LIN {X -0.064,Y -285.308,Z 785.698,A 0.000,B 0.000,C 90.000,E1 305.598} C_DIS
LIN {X 0.000,Y -296.735,Z 785.683,A 0.000,B 0.000,C 90.000,E1 302.880} C_DIS
LIN {X -0.130,Y -309.503,Z 785.668,A 0.000,B 0.000,C 90.000,E1 300.256} C_DIS
LIN {X -0.044,Y -325.399,Z 785.652,A 0.000,B 0.000,C 90.000,E1 297.334} C_DIS
LIN {X -0.084,Y -344.528,Z 785.634,A 0.000,B 0.000,C 90.000,E1 294.207} C_DIS
LIN {X 0.058,Y -365.735,Z 785.618,A 0.000,B 0.000,C 90.000,E1 291.153} C_DIS
LIN {X 0.141,Y -382.144,Z 785.606,A 0.000,B 0.000,C 90.000,E1 289.087} C_DIS
LIN {X 0.210,Y -399.426,Z 785.595,A 0.000,B 0.000,C 90.000,E1 287.094} C_DIS
LIN {X -0.176,Y -414.390,Z 785.586,A 0.000,B 0.000,C 90.000,E1 285.481} C_DIS
LIN {X 0.184,Y -426.696,Z 785.578,A 0.000,B 0.000,C 90.000,E1 284.064} C_DIS
LIN {X -0.207,Y -438.621,Z 785.571,A 0.000,B 0.000,C 90.000,E1 282.771} C_DIS
LIN {X -0.227,Y -447.840,Z 785.565,A 0.000,B 0.000,C 90.000,E1 281.715} C_DIS
LIN {X -0.140,Y -456.433,Z 785.559,A 0.000,B 0.000,C 90.000,E1 280.658} C_DIS
LIN {X -0.035,Y -464.422,Z 785.553,A 0.000,B 0.000,C 90.000,E1 279.613} C_DIS
LIN {X 0.170,Y -471.836,Z 785.548,A 0.000,B 0.000,C 90.000,E1 278.568} C_DIS
LIN {X 0.131,Y -476.934,Z 785.544,A 0.000,B 0.000,C 90.000,E1 277.814} C_DIS
LIN {X 0.070,Y -481.460,Z 785.539,A 0.000,B 0.000,C 90.000,E1 277.068} C_DIS
LIN {X 0.114,Y -485.271,Z 785.535,A 0.000,B 0.000,C 90.000,E1 276.315} C_DIS
LIN {X 0.133,Y -488.291,Z 785.531,A 0.000,B 0.000,C 90.000,E1 275.568} C_DIS
LIN {X -0.152,Y -489.902,Z 785.528,A 0.000,B 0.000,C 90.000,E1 275.106} C_DIS
LIN {X 0.059,Y -491.124,Z 785.526,A 0.000,B 0.000,C 90.000,E1 274.588} C_DIS
LIN {X -0.247,Y -491.992,Z 785.523,A 0.000,B 0.000,C 90.000,E1 274.131} C_DIS
LIN {X -0.020,Y -492.449,Z 785.520,A 0.000,B 0.000,C 90.000,E1 273.612} C_DIS
LIN {X 0.209,Y -492.461,Z 785.517,A 0.000,B 0.000,C 90.000,E1 273.094} C_DIS
LIN {X -0.078,Y -492.080,Z 785.515,A 0.000,B 0.000,C 90.000,E1 272.636} C_DIS
LIN {X 0.129,Y -491.280,Z 785.512,A 0.000,B 0.000,C 90.000,E1 272.121} C_DIS
LIN {X -0.139,Y -490.046,Z 785.509,A 0.000,B 0.000,C 90.000,E1 271.661} C_DIS
LIN {X 0.060,Y -488.375,Z 785.506,A 0.000,B 0.000,C 90.000,E1 271.146} C_DIS
LIN {X -0.232,Y -486.237,Z 785.504,A 0.000,B 0.000,C 90.000,E1 270.688} C_DIS
LIN {X -0.047,Y -483.535,Z 785.501,A 0.000,B 0.000,C 90.000,E1 270.172} C_DIS
LIN {X 0.118,Y -480.277,Z 785.498,A 0.000,B 0.000,C 90.000,E1 269.656} C_DIS
LIN {X -0.214,Y -476.251,Z 785.495,A 0.000,B 0.000,C 90.000,E1 269.198} C_DIS
LIN {X -0.089,Y -471.307,Z 785.493,A 0.000,B 0.000,C 90.000,E1 268.682} C_DIS
LIN {X 0.184,Y -465.469,Z 785.490,A 0.000,B 0.000,C 90.000,E1 268.167} C_DIS
LIN {X -0.118,Y -462.390,Z 785.489,A 0.000,B 0.000,C 90.000,E1 267.993} C_DIS
LIN {X 0.027,Y -458.873,Z 785.488,A 0.000,B 0.000,C 90.000,E1 267.764} C_DIS
LIN {X 0.008,Y -451.802,Z 785.486,A 0.000,B 0.000,C 90.000,E1 267.421} C_DIS
LIN {X 0.059,Y -444.230,Z 785.484,A 0.000,B 0.000,C 90.000,E1 267.135} C_DIS
LIN {X 0.195,Y -436.200,Z 785.483,A 0.000,B 0.000,C 90.000,E1 266.906} C_DIS
LIN {X 0.089,Y -432.234,Z 785.483,A 0.000,B 0.000,C 90.000,E1 266.846} C_DIS
LIN {X -0.201,Y -423.188,Z 785.482,A 0.000,B 0.000,C 90.000,E1 266.788} C_DIS
LIN {X 0.060,Y -417.117,Z 785.482,A 0.000,B 0.000,C 90.000,E1 266.731} C_DIS
LIN {X -0.009,Y -180.966,Z 785.482,A 0.000,B 0.000,C 90.000,E1 266.731} C_DIS
LIN {X 0.007,Y -180.865,Z 785.472,A 0.000,B 0.000,C 90.000,E1 265.008} C_DIS
LIN {X 0.060,Y -178.978,Z 785.444,A 0.000,B 0.000,C 90.000,E1 259.926} C_DIS
LIN {X 0.069,Y -177.945,Z 785.435,A 0.000,B 0.000,C 90.000,E1 258.229} C_DIS
LIN {X 0.084,Y -175.585,Z 785.411,A 0.000,B 0.000,C 90.000,E1 253.976} C_DIS
LIN {X -0.072,Y -172.311,Z 785.387,A 0.000,B 0.000,C 90.000,E1 249.752} C_DIS
LIN {X -0.093,Y -171.789,Z 785.383,A 0.000,B 0.000,C 90.000,E1 248.901} C_DIS
LIN {X -0.055,Y -169.458,Z 785.368,A 0.000,B 0.000,C 90.000,E1 246.305} C_DIS
LIN {X 0.001,Y -166.786,Z 785.349,A 0.000,B 0.000,C 90.000,E1 242.820} C_DIS
LIN {X -0.003,Y -162.767,Z 785.325,A 0.000,B 0.000,C 90.000,E1 238.456} C_DIS
LIN {X -0.027,Y -161.456,Z 785.315,A 0.000,B 0.000,C 90.000,E1 236.707} C_DIS
LIN {X 0.015,Y -157.450,Z 785.290,A 0.000,B 0.000,C 90.000,E1 232.271} C_DIS
LIN {X -0.053,Y -155.460,Z 785.276,A 0.000,B 0.000,C 90.000,E1 229.622} C_DIS
LIN {X -0.011,Y -151.774,Z 785.251,A 0.000,B 0.000,C 90.000,E1 225.121} C_DIS
LIN {X 0.006,Y -149.980,Z 785.236,A 0.000,B 0.000,C 90.000,E1 222.405} C_DIS
LIN {X -0.074,Y -146.815,Z 785.210,A 0.000,B 0.000,C 90.000,E1 217.890} C_DIS
LIN {X 0.033,Y -145.392,Z 785.195,A 0.000,B 0.000,C 90.000,E1 215.105} C_DIS
LIN {X -0.049,Y -142.828,Z 785.170,A 0.000,B 0.000,C 90.000,E1 210.541} C_DIS
LIN {X 0.007,Y -141.441,Z 785.149,A 0.000,B 0.000,C 90.000,E1 206.821} C_DIS
LIN {X 0.052,Y -139.368,Z 785.113,A 0.000,B 0.000,C 90.000,E1 200.301} C_DIS
LIN {X 0.038,Y -138.815,Z 785.097,A 0.000,B 0.000,C 90.000,E1 197.511} C_DIS
LIN {X -0.048,Y -138.352,Z 785.056,A 0.000,B 0.000,C 90.000,E1 190.074} C_DIS
LIN {X 0.065,Y -139.537,Z 785.004,A 0.000,B 0.000,C 90.000,E1 180.688} C_DIS
LIN {X 0.018,Y -141.227,Z 784.973,A 0.000,B 0.000,C 90.000,E1 175.122} C_DIS
LIN {X -0.023,Y -142.599,Z 784.957,A 0.000,B 0.000,C 90.000,E1 172.356} C_DIS
LIN {X 0.071,Y -144.904,Z 784.932,A 0.000,B 0.000,C 90.000,E1 167.701} C_DIS
LIN {X 0.024,Y -147.533,Z 784.911,A 0.000,B 0.000,C 90.000,E1 164.047} C_DIS
LIN {X -0.044,Y -150.131,Z 784.891,A 0.000,B 0.000,C 90.000,E1 160.423} C_DIS
LIN {X -0.033,Y -153.496,Z 784.871,A 0.000,B 0.000,C 90.000,E1 156.794} C_DIS
LIN {X 0.030,Y -157.861,Z 784.846,A 0.000,B 0.000,C 90.000,E1 152.281} C_DIS
LIN {X -0.014,Y -162.146,Z 784.826,A 0.000,B 0.000,C 90.000,E1 148.742} C_DIS
LIN {X -0.036,Y -166.352,Z 784.807,A 0.000,B 0.000,C 90.000,E1 145.229} C_DIS
LIN {X -0.030,Y -171.368,Z 784.787,A 0.000,B 0.000,C 90.000,E1 141.743} C_DIS
LIN {X -0.103,Y -176.276,Z 784.768,A 0.000,B 0.000,C 90.000,E1 138.324} C_DIS
LIN {X 0.015,Y -180.561,Z 784.754,A 0.000,B 0.000,C 90.000,E1 135.729} C_DIS
LIN {X -0.007,Y -185.963,Z 784.735,A 0.000,B 0.000,C 90.000,E1 132.366} C_DIS
LIN {X 0.050,Y -190.594,Z 784.721,A 0.000,B 0.000,C 90.000,E1 129.850} C_DIS
LIN {X 0.040,Y -192.511,Z 784.715,A 0.000,B 0.000,C 90.000,E1 128.705} C_DIS
LIN {X 0.013,Y -292.777,Z 784.715,A 0.000,B 0.000,C 90.000,E1 128.705} C_DIS
LIN {X -0.041,Y -298.777,Z 784.714,A 0.000,B 0.000,C 90.000,E1 128.463} C_DIS
LIN {X -0.049,Y -301.480,Z 784.712,A 0.000,B 0.000,C 90.000,E1 128.222} C_DIS
LIN {X 0.044,Y -305.237,Z 784.709,A 0.000,B 0.000,C 90.000,E1 127.684} C_DIS
LIN {X -0.001,Y -306.900,Z 784.708,A 0.000,B 0.000,C 90.000,E1 127.363} C_DIS
LIN {X 0.010,Y -308.204,Z 784.706,A 0.000,B 0.000,C 90.000,E1 127.030} C_DIS
LIN {X -0.126,Y -320.271,Z 784.684,A 0.000,B 0.000,C 90.000,E1 123.166} C_DIS
LIN {X 0.162,Y -330.699,Z 784.668,A 0.000,B 0.000,C 90.000,E1 120.256} C_DIS
LIN {X 0.095,Y -342.483,Z 784.653,A 0.000,B 0.000,C 90.000,E1 117.462} C_DIS
LIN {X 0.063,Y -355.724,Z 784.637,A 0.000,B 0.000,C 90.000,E1 114.719} C_DIS
LIN {X 0.022,Y -368.815,Z 784.624,A 0.000,B 0.000,C 90.000,E1 112.333} C_DIS
LIN {X 0.017,Y -383.245,Z 784.611,A 0.000,B 0.000,C 90.000,E1 109.993} C_DIS
LIN {X 0.111,Y -399.118,Z 784.598,A 0.000,B 0.000,C 90.000,E1 107.692} C_DIS
LIN {X -0.026,Y -416.549,Z 784.586,A 0.000,B 0.000,C 90.000,E1 105.481} C_DIS
LIN {X 0.065,Y -435.644,Z 784.574,A 0.000,B 0.000,C 90.000,E1 103.300} C_DIS
LIN {X -0.186,Y -455.766,Z 784.563,A 0.000,B 0.000,C 90.000,E1 101.299} C_DIS
LIN {X 0.127,Y -468.504,Z 784.556,A 0.000,B 0.000,C 90.000,E1 100.074} C_DIS
LIN {X 0.016,Y -470.441,Z 784.555,A 0.000,B 0.000,C 90.000,E1 99.849} C_DIS
LIN {X -0.014,Y -471.912,Z 784.553,A 0.000,B 0.000,C 90.000,E1 99.613} C_DIS
LIN {X 0.087,Y -473.945,Z 784.551,A 0.000,B 0.000,C 90.000,E1 99.095} C_DIS
LIN {X -0.198,Y -474.842,Z 784.548,A 0.000,B 0.000,C 90.000,E1 98.624} C_DIS
LIN {X -0.076,Y -474.760,Z 784.545,A 0.000,B 0.000,C 90.000,E1 98.106} C_DIS
LIN {X 0.054,Y -473.694,Z 784.542,A 0.000,B 0.000,C 90.000,E1 97.587} C_DIS
LIN {X -0.085,Y -472.745,Z 784.541,A 0.000,B 0.000,C 90.000,E1 97.352} C_DIS
LIN {X 0.186,Y -471.459,Z 784.539,A 0.000,B 0.000,C 90.000,E1 97.068} C_DIS
LIN {X -0.107,Y -453.695,Z 784.524,A 0.000,B 0.000,C 90.000,E1 94.302} C_DIS
LIN {X 0.040,Y -443.147,Z 784.514,A 0.000,B 0.000,C 90.000,E1 92.465} C_DIS
LIN {X -0.210,Y -433.992,Z 784.505,A 0.000,B 0.000,C 90.000,E1 90.917} C_DIS
LIN {X -0.191,Y -424.524,Z 784.496,A 0.000,B 0.000,C 90.000,E1 89.312} C_DIS
LIN {X 0.088,Y -414.894,Z 784.487,A 0.000,B 0.000,C 90.000,E1 87.650} C_DIS
LIN {X -0.132,Y -403.562,Z 784.476,A 0.000,B 0.000,C 90.000,E1 85.755} C_DIS
LIN {X -0.143,Y -392.119,Z 784.465,A 0.000,B 0.000,C 90.000,E1 83.799} C_DIS
LIN {X 0.096,Y -376.284,Z 784.450,A 0.000,B 0.000,C 90.000,E1 80.905} C_DIS
LIN {X 0.002,Y -362.489,Z 784.435,A 0.000,B 0.000,C 90.000,E1 78.285} C_DIS
LIN {X 0.095,Y -350.867,Z 784.422,A 0.000,B 0.000,C 90.000,E1 75.880} C_DIS
LIN {X 0.065,Y -339.326,Z 784.408,A 0.000,B 0.000,C 90.000,E1 73.449} C_DIS
LIN {X 0.055,Y -328.066,Z 784.394,A 0.000,B 0.000,C 90.000,E1 70.967} C_DIS
LIN {X -0.107,Y -317.052,Z 784.380,A 0.000,B 0.000,C 90.000,E1 68.465} C_DIS
LIN {X -0.057,Y -302.829,Z 784.360,A 0.000,B 0.000,C 90.000,E1 64.897} C_DIS
LIN {X -0.102,Y -289.904,Z 784.340,A 0.000,B 0.000,C 90.000,E1 61.257} C_DIS
LIN {X -0.056,Y -280.077,Z 784.323,A 0.000,B 0.000,C 90.000,E1 58.201} C_DIS
LIN {X -0.139,Y -271.759,Z 784.308,A 0.000,B 0.000,C 90.000,E1 55.468} C_DIS
LIN {X 0.049,Y -265.658,Z 784.296,A 0.000,B 0.000,C 90.000,E1 53.336} C_DIS
LIN {X -0.092,Y -259.561,Z 784.285,A 0.000,B 0.000,C 90.000,E1 51.251} C_DIS
LIN {X 0.013,Y -251.506,Z 784.269,A 0.000,B 0.000,C 90.000,E1 48.366} C_DIS
LIN {X -0.117,Y -241.907,Z 784.248,A 0.000,B 0.000,C 90.000,E1 44.757} C_DIS
LIN {X -0.069,Y -236.363,Z 784.236,A 0.000,B 0.000,C 90.000,E1 42.528} C_DIS
LIN {X 0.039,Y -227.342,Z 784.215,A 0.000,B 0.000,C 90.000,E1 38.749} C_DIS
LIN {X -0.030,Y -218.837,Z 784.194,A 0.000,B 0.000,C 90.000,E1 34.945} C_DIS
LIN {X -0.017,Y -211.028,Z 784.172,A 0.000,B 0.000,C 90.000,E1 31.052} C_DIS
LIN {X -0.029,Y -205.490,Z 784.155,A 0.000,B 0.000,C 90.000,E1 27.897} C_DIS
LIN {X -0.006,Y -200.725,Z 784.137,A 0.000,B 0.000,C 90.000,E1 24.695} C_DIS
LIN {X -0.035,Y -195.745,Z 784.115,A 0.000,B 0.000,C 90.000,E1 20.663} C_DIS
LIN {X 0.009,Y -191.908,Z 784.092,A 0.000,B 0.000,C 90.000,E1 16.567} C_DIS
LIN {X -0.103,Y -188.694,Z 784.065,A 0.000,B 0.000,C 90.000,E1 11.658} C_DIS
LIN {X 0.003,Y -186.624,Z 784.018,A 0.000,B 0.000,C 90.000,E1 3.326} C_DIS
LIN {X 0.001,Y -188.497,Z 783.970,A 0.000,B 0.000,C 90.000,E1 354.546} C_DIS
LIN {X 0.004,Y -192.032,Z 783.938,A 0.000,B 0.000,C 90.000,E1 348.757} C_DIS
LIN {X 0.089,Y -195.633,Z 783.915,A 0.000,B 0.000,C 90.000,E1 344.629} C_DIS
LIN {X -0.062,Y -200.258,Z 783.892,A 0.000,B 0.000,C 90.000,E1 340.604} C_DIS
LIN {X 0.083,Y -205.972,Z 783.870,A 0.000,B 0.000,C 90.000,E1 336.538} C_DIS
LIN {X -0.024,Y -211.217,Z 783.852,A 0.000,B 0.000,C 90.000,E1 333.384} C_DIS
LIN {X -0.038,Y -218.499,Z 783.830,A 0.000,B 0.000,C 90.000,E1 329.459} C_DIS
LIN {X 0.036,Y -224.827,Z 783.813,A 0.000,B 0.000,C 90.000,E1 326.342} C_DIS
LIN {X -0.086,Y -233.389,Z 783.792,A 0.000,B 0.000,C 90.000,E1 322.557} C_DIS
LIN {X 0.078,Y -242.712,Z 783.771,A 0.000,B 0.000,C 90.000,E1 318.771} C_DIS
LIN {X -0.015,Y -252.902,Z 783.751,A 0.000,B 0.000,C 90.000,E1 315.121} C_DIS
LIN {X 0.002,Y -262.764,Z 783.733,A 0.000,B 0.000,C 90.000,E1 311.881} C_DIS
LIN {X -0.116,Y -274.750,Z 783.713,A 0.000,B 0.000,C 90.000,E1 308.382} C_DIS
LIN {X 0.093,Y -288.032,Z 783.694,A 0.000,B 0.000,C 90.000,E1 304.898} C_DIS
LIN {X 0.064,Y -298.190,Z 783.681,A 0.000,B 0.000,C 90.000,E1 302.546} C_DIS
LIN {X -0.026,Y -311.133,Z 783.666,A 0.000,B 0.000,C 90.000,E1 299.922} C_DIS
LIN {X 0.119,Y -327.130,Z 783.650,A 0.000,B 0.000,C 90.000,E1 297.001} C_DIS
LIN {X -0.012,Y -344.443,Z 783.634,A 0.000,B 0.000,C 90.000,E1 294.207} C_DIS
LIN {X 0.070,Y -363.354,Z 783.619,A 0.000,B 0.000,C 90.000,E1 291.461} C_DIS
LIN {X 0.060,Y -379.537,Z 783.608,A 0.000,B 0.000,C 90.000,E1 289.396} C_DIS
LIN {X 0.094,Y -399.416,Z 783.595,A 0.000,B 0.000,C 90.000,E1 287.094} C_DIS
LIN {X 0.035,Y -414.432,Z 783.586,A 0.000,B 0.000,C 90.000,E1 285.426} C_DIS
LIN {X 0.047,Y -426.654,Z 783.578,A 0.000,B 0.000,C 90.000,E1 284.064} C_DIS
LIN {X 0.079,Y -438.510,Z 783.571,A 0.000,B 0.000,C 90.000,E1 282.715} C_DIS
LIN {X 0.066,Y -447.727,Z 783.565,A 0.000,B 0.000,C 90.000,E1 281.658} C_DIS
LIN {X 0.159,Y -456.331,Z 783.559,A 0.000,B 0.000,C 90.000,E1 280.602} C_DIS
LIN {X -0.189,Y -464.285,Z 783.553,A 0.000,B 0.000,C 90.000,E1 279.613} C_DIS
LIN {X 0.012,Y -471.747,Z 783.548,A 0.000,B 0.000,C 90.000,E1 278.568} C_DIS
LIN {X -0.237,Y -478.485,Z 783.542,A 0.000,B 0.000,C 90.000,E1 277.587} C_DIS
LIN {X -0.221,Y -482.779,Z 783.538,A 0.000,B 0.000,C 90.000,E1 276.834} C_DIS
LIN {X -0.229,Y -486.319,Z 783.534,A 0.000,B 0.000,C 90.000,E1 276.087} C_DIS
LIN {X -0.033,Y -488.289,Z 783.531,A 0.000,B 0.000,C 90.000,E1 275.568} C_DIS
LIN {X 0.169,Y -489.900,Z 783.528,A 0.000,B 0.000,C 90.000,E1 275.049} C_DIS
LIN {X -0.107,Y -491.132,Z 783.525,A 0.000,B 0.000,C 90.000,E1 274.588} C_DIS
LIN {X 0.077,Y -491.995,Z 783.523,A 0.000,B 0.000,C 90.000,E1 274.073} C_DIS
LIN {X -0.187,Y -492.450,Z 783.520,A 0.000,B 0.000,C 90.000,E1 273.612} C_DIS
LIN {X 0.042,Y -492.493,Z 783.517,A 0.000,B 0.000,C 90.000,E1 273.094} C_DIS
LIN {X 0.246,Y -492.142,Z 783.514,A 0.000,B 0.000,C 90.000,E1 272.579} C_DIS
LIN {X -0.038,Y -491.332,Z 783.512,A 0.000,B 0.000,C 90.000,E1 272.121} C_DIS
LIN {X 0.184,Y -490.093,Z 783.509,A 0.000,B 0.000,C 90.000,E1 271.604} C_DIS
LIN {X -0.104,Y -488.417,Z 783.506,A 0.000,B 0.000,C 90.000,E1 271.146} C_DIS
LIN {X 0.090,Y -486.263,Z 783.504,A 0.000,B 0.000,C 90.000,E1 270.630} C_DIS
LIN {X -0.210,Y -483.566,Z 783.501,A 0.000,B 0.000,C 90.000,E1 270.172} C_DIS
LIN {X -0.044,Y -480.305,Z 783.498,A 0.000,B 0.000,C 90.000,E1 269.656} C_DIS
LIN {X 0.102,Y -476.248,Z 783.495,A 0.000,B 0.000,C 90.000,E1 269.141} C_DIS
LIN {X -0.073,Y -473.928,Z 783.494,A 0.000,B 0.000,C 90.000,E1 268.912} C_DIS
LIN {X 0.158,Y -468.582,Z 783.491,A 0.000,B 0.000,C 90.000,E1 268.396} C_DIS
LIN {X 0.107,Y -465.525,Z 783.490,A 0.000,B 0.000,C 90.000,E1 268.165} C_DIS
LIN {X -0.198,Y -462.443,Z 783.489,A 0.000,B 0.000,C 90.000,E1 267.993} C_DIS
LIN {X -0.033,Y -455.738,Z 783.487,A 0.000,B 0.000,C 90.000,E1 267.593} C_DIS
LIN {X -0.218,Y -448.581,Z 783.485,A 0.000,B 0.000,C 90.000,E1 267.306} C_DIS
LIN {X 0.097,Y -440.943,Z 783.484,A 0.000,B 0.000,C 90.000,E1 267.020} C_DIS
LIN {X 0.036,Y -432.403,Z 783.482,A 0.000,B 0.000,C 90.000,E1 266.846} C_DIS
LIN {X 0.149,Y -423.558,Z 783.482,A 0.000,B 0.000,C 90.000,E1 266.731} C_DIS
LIN {X -0.020,Y -418.188,Z 783.482,A 0.000,B 0.000,C 90.000,E1 266.731} C_DIS
LIN {X -0.045,Y -180.965,Z 783.482,A 0.000,B 0.000,C 90.000,E1 266.731} C_DIS
LIN {X -0.035,Y -180.861,Z 783.472,A 0.000,B 0.000,C 90.000,E1 265.008} C_DIS
LIN {X 0.019,Y -178.974,Z 783.444,A 0.000,B 0.000,C 90.000,E1 259.926} C_DIS
LIN {X 0.029,Y -177.936,Z 783.435,A 0.000,B 0.000,C 90.000,E1 258.229} C_DIS
LIN {X 0.044,Y -175.575,Z 783.411,A 0.000,B 0.000,C 90.000,E1 253.976} C_DIS
LIN {X 0.051,Y -172.303,Z 783.387,A 0.000,B 0.000,C 90.000,E1 249.699} C_DIS
LIN {X 0.028,Y -171.781,Z 783.383,A 0.000,B 0.000,C 90.000,E1 248.847} C_DIS
LIN {X 0.000,Y -168.712,Z 783.363,A 0.000,B 0.000,C 90.000,E1 245.409} C_DIS
LIN {X 0.039,Y -166.776,Z 783.349,A 0.000,B 0.000,C 90.000,E1 242.794} C_DIS
LIN {X -0.041,Y -162.756,Z 783.325,A 0.000,B 0.000,C 90.000,E1 238.456} C_DIS
LIN {X -0.065,Y -161.446,Z 783.315,A 0.000,B 0.000,C 90.000,E1 236.707} C_DIS
LIN {X -0.024,Y -157.439,Z 783.290,A 0.000,B 0.000,C 90.000,E1 232.271} C_DIS
LIN {X 0.011,Y -155.447,Z 783.276,A 0.000,B 0.000,C 90.000,E1 229.585} C_DIS
LIN {X 0.059,Y -151.766,Z 783.251,A 0.000,B 0.000,C 90.000,E1 225.081} C_DIS
LIN {X 0.070,Y -149.968,Z 783.236,A 0.000,B 0.000,C 90.000,E1 222.366} C_DIS
LIN {X -0.019,Y -146.806,Z 783.210,A 0.000,B 0.000,C 90.000,E1 217.855} C_DIS
LIN {X -0.003,Y -145.383,Z 783.195,A 0.000,B 0.000,C 90.000,E1 215.105} C_DIS
LIN {X -0.011,Y -142.442,Z 783.164,A 0.000,B 0.000,C 90.000,E1 209.589} C_DIS
LIN {X 0.036,Y -141.434,Z 783.149,A 0.000,B 0.000,C 90.000,E1 206.796} C_DIS
LIN {X 0.017,Y -139.366,Z 783.113,A 0.000,B 0.000,C 90.000,E1 200.301} C_DIS
LIN {X 0.003,Y -138.813,Z 783.097,A 0.000,B 0.000,C 90.000,E1 197.511} C_DIS
LIN {X 0.054,Y -138.351,Z 783.056,A 0.000,B 0.000,C 90.000,E1 190.018} C_DIS
LIN {X 0.030,Y -139.539,Z 783.004,A 0.000,B 0.000,C 90.000,E1 180.688} C_DIS
LIN {X -0.018,Y -141.233,Z 782.973,A 0.000,B 0.000,C 90.000,E1 175.122} C_DIS
LIN {X -0.059,Y -142.604,Z 782.957,A 0.000,B 0.000,C 90.000,E1 172.356} C_DIS
LIN {X 0.035,Y -144.913,Z 782.932,A 0.000,B 0.000,C 90.000,E1 167.701} C_DIS
LIN {X 0.028,Y -147.542,Z 782.911,A 0.000,B 0.000,C 90.000,E1 164.031} C_DIS
LIN {X 0.061,Y -150.143,Z 782.891,A 0.000,B 0.000,C 90.000,E1 160.369} C_DIS
LIN {X -0.070,Y -153.511,Z 782.871,A 0.000,B 0.000,C 90.000,E1 156.794} C_DIS
LIN {X -0.007,Y -157.876,Z 782.846,A 0.000,B 0.000,C 90.000,E1 152.281} C_DIS
LIN {X -0.052,Y -162.163,Z 782.826,A 0.000,B 0.000,C 90.000,E1 148.742} C_DIS
LIN {X 0.062,Y -166.369,Z 782.807,A 0.000,B 0.000,C 90.000,E1 145.182} C_DIS
LIN {X 0.065,Y -171.386,Z 782.787,A 0.000,B 0.000,C 90.000,E1 141.698} C_DIS
LIN {X 0.105,Y -176.296,Z 782.768,A 0.000,B 0.000,C 90.000,E1 138.243} C_DIS
LIN {X -0.027,Y -180.583,Z 782.754,A 0.000,B 0.000,C 90.000,E1 135.729} C_DIS
LIN {X -0.048,Y -185.985,Z 782.735,A 0.000,B 0.000,C 90.000,E1 132.366} C_DIS
LIN {X 0.007,Y -190.619,Z 782.721,A 0.000,B 0.000,C 90.000,E1 129.850} C_DIS
LIN {X -0.066,Y -192.489,Z 782.715,A 0.000,B 0.000,C 90.000,E1 128.749} C_DIS
LIN {X -0.136,Y -292.326,Z 782.715,A 0.000,B 0.000,C 90.000,E1 128.749} C_DIS
LIN {X 0.085,Y -294.367,Z 782.715,A 0.000,B 0.000,C 90.000,E1 128.669} C_DIS
LIN {X -0.106,Y -299.048,Z 782.714,A 0.000,B 0.000,C 90.000,E1 128.463} C_DIS
LIN {X 0.122,Y -301.653,Z 782.712,A 0.000,B 0.000,C 90.000,E1 128.177} C_DIS
LIN {X 0.079,Y -305.413,Z 782.709,A 0.000,B 0.000,C 90.000,E1 127.649} C_DIS
LIN {X 0.090,Y -307.024,Z 782.707,A 0.000,B 0.000,C 90.000,E1 127.317} C_DIS
LIN {X 0.043,Y -308.289,Z 782.706,A 0.000,B 0.000,C 90.000,E1 126.996} C_DIS
LIN {X 0.162,Y -320.344,Z 782.684,A 0.000,B 0.000,C 90.000,E1 123.086} C_DIS
LIN {X 0.005,Y -330.785,Z 782.668,A 0.000,B 0.000,C 90.000,E1 120.256} C_DIS
LIN {X -0.066,Y -342.583,Z 782.653,A 0.000,B 0.000,C 90.000,E1 117.462} C_DIS
LIN {X -0.102,Y -355.838,Z 782.637,A 0.000,B 0.000,C 90.000,E1 114.719} C_DIS
LIN {X -0.146,Y -368.942,Z 782.624,A 0.000,B 0.000,C 90.000,E1 112.333} C_DIS
LIN {X -0.154,Y -383.387,Z 782.611,A 0.000,B 0.000,C 90.000,E1 109.993} C_DIS
LIN {X -0.063,Y -399.278,Z 782.598,A 0.000,B 0.000,C 90.000,E1 107.692} C_DIS
LIN {X 0.197,Y -416.726,Z 782.586,A 0.000,B 0.000,C 90.000,E1 105.426} C_DIS
LIN {X -0.115,Y -435.837,Z 782.574,A 0.000,B 0.000,C 90.000,E1 103.300} C_DIS
LIN {X 0.086,Y -455.967,Z 782.563,A 0.000,B 0.000,C 90.000,E1 101.243} C_DIS
LIN {X -0.044,Y -468.675,Z 782.556,A 0.000,B 0.000,C 90.000,E1 100.074} C_DIS
LIN {X -0.170,Y -470.586,Z 782.555,A 0.000,B 0.000,C 90.000,E1 99.849} C_DIS
LIN {X -0.217,Y -472.037,Z 782.553,A 0.000,B 0.000,C 90.000,E1 99.613} C_DIS
LIN {X -0.116,Y -474.018,Z 782.550,A 0.000,B 0.000,C 90.000,E1 99.095} C_DIS
LIN {X 0.069,Y -474.873,Z 782.548,A 0.000,B 0.000,C 90.000,E1 98.568} C_DIS
LIN {X 0.192,Y -474.754,Z 782.545,A 0.000,B 0.000,C 90.000,E1 98.049} C_DIS
LIN {X -0.146,Y -473.645,Z 782.542,A 0.000,B 0.000,C 90.000,E1 97.587} C_DIS
LIN {X 0.184,Y -472.671,Z 782.541,A 0.000,B 0.000,C 90.000,E1 97.296} C_DIS
LIN {X -0.015,Y -471.355,Z 782.539,A 0.000,B 0.000,C 90.000,E1 97.068} C_DIS
LIN {X 0.150,Y -453.580,Z 782.524,A 0.000,B 0.000,C 90.000,E1 94.245} C_DIS
LIN {X -0.153,Y -443.023,Z 782.514,A 0.000,B 0.000,C 90.000,E1 92.465} C_DIS
LIN {X 0.032,Y -433.887,Z 782.505,A 0.000,B 0.000,C 90.000,E1 90.859} C_DIS
LIN {X 0.044,Y -424.425,Z 782.496,A 0.000,B 0.000,C 90.000,E1 89.255} C_DIS
LIN {X -0.006,Y -413.178,Z 782.485,A 0.000,B 0.000,C 90.000,E1 87.364} C_DIS
LIN {X 0.087,Y -403.472,Z 782.476,A 0.000,B 0.000,C 90.000,E1 85.698} C_DIS
LIN {X 0.077,Y -390.407,Z 782.464,A 0.000,B 0.000,C 90.000,E1 83.457} C_DIS
LIN {X -0.079,Y -376.210,Z 782.449,A 0.000,B 0.000,C 90.000,E1 80.905} C_DIS
LIN {X 0.162,Y -360.948,Z 782.433,A 0.000,B 0.000,C 90.000,E1 77.937} C_DIS
LIN {X -0.045,Y -349.388,Z 782.420,A 0.000,B 0.000,C 90.000,E1 75.574} C_DIS
LIN {X -0.098,Y -337.880,Z 782.406,A 0.000,B 0.000,C 90.000,E1 73.142} C_DIS
LIN {X 0.178,Y -326.659,Z 782.392,A 0.000,B 0.000,C 90.000,E1 70.604} C_DIS
LIN {X -0.095,Y -314.404,Z 782.377,A 0.000,B 0.000,C 90.000,E1 67.794} C_DIS
LIN {X -0.012,Y -300.461,Z 782.357,A 0.000,B 0.000,C 90.000,E1 64.204} C_DIS
LIN {X -0.009,Y -287.816,Z 782.336,A 0.000,B 0.000,C 90.000,E1 60.539} C_DIS
LIN {X 0.135,Y -278.207,Z 782.319,A 0.000,B 0.000,C 90.000,E1 57.454} C_DIS
LIN {X 0.152,Y -269.987,Z 782.304,A 0.000,B 0.000,C 90.000,E1 54.689} C_DIS
LIN {X 0.059,Y -261.882,Z 782.288,A 0.000,B 0.000,C 90.000,E1 51.904} C_DIS
LIN {X 0.053,Y -253.846,Z 782.273,A 0.000,B 0.000,C 90.000,E1 49.057} C_DIS
LIN {X -0.001,Y -244.130,Z 782.253,A 0.000,B 0.000,C 90.000,E1 45.445} C_DIS
LIN {X -0.133,Y -236.699,Z 782.236,A 0.000,B 0.000,C 90.000,E1 42.528} C_DIS
LIN {X -0.012,Y -227.656,Z 782.215,A 0.000,B 0.000,C 90.000,E1 38.749} C_DIS
LIN {X -0.071,Y -219.130,Z 782.194,A 0.000,B 0.000,C 90.000,E1 34.945} C_DIS
LIN {X -0.048,Y -211.314,Z 782.172,A 0.000,B 0.000,C 90.000,E1 31.052} C_DIS
LIN {X -0.051,Y -205.757,Z 782.155,A 0.000,B 0.000,C 90.000,E1 27.897} C_DIS
LIN {X -0.045,Y -199.916,Z 782.133,A 0.000,B 0.000,C 90.000,E1 23.898} C_DIS
LIN {X 0.090,Y -195.141,Z 782.110,A 0.000,B 0.000,C 90.000,E1 19.812} C_DIS
LIN {X 0.058,Y -191.502,Z 782.088,A 0.000,B 0.000,C 90.000,E1 15.733} C_DIS
LIN {X 0.072,Y -188.523,Z 782.060,A 0.000,B 0.000,C 90.000,E1 10.782} C_DIS
LIN {X -0.029,Y -187.969,Z 781.979,A 0.000,B 0.000,C 90.000,E1 356.216} C_DIS
LIN {X 0.080,Y -190.984,Z 781.947,A 0.000,B 0.000,C 90.000,E1 350.387} C_DIS
LIN {X 0.049,Y -194.962,Z 781.919,A 0.000,B 0.000,C 90.000,E1 345.463} C_DIS
LIN {X 0.002,Y -199.392,Z 781.897,A 0.000,B 0.000,C 90.000,E1 341.402} C_DIS
LIN {X 0.040,Y -204.919,Z 781.874,A 0.000,B 0.000,C 90.000,E1 337.358} C_DIS
LIN {X 0.095,Y -209.981,Z 781.857,A 0.000,B 0.000,C 90.000,E1 334.152} C_DIS
LIN {X -0.060,Y -217.120,Z 781.835,A 0.000,B 0.000,C 90.000,E1 330.255} C_DIS
LIN {X 0.045,Y -223.348,Z 781.817,A 0.000,B 0.000,C 90.000,E1 327.120} C_DIS
LIN {X 0.057,Y -231.725,Z 781.796,A 0.000,B 0.000,C 90.000,E1 323.290} C_DIS
LIN {X 0.013,Y -240.884,Z 781.775,A 0.000,B 0.000,C 90.000,E1 319.542} C_DIS
LIN {X 0.036,Y -249.821,Z 781.757,A 0.000,B 0.000,C 90.000,E1 316.215} C_DIS
LIN {X -0.004,Y -260.516,Z 781.737,A 0.000,B 0.000,C 90.000,E1 312.609} C_DIS
LIN {X -0.012,Y -272.284,Z 781.717,A 0.000,B 0.000,C 90.000,E1 309.072} C_DIS
LIN {X -0.005,Y -282.531,Z 781.702,A 0.000,B 0.000,C 90.000,E1 306.297} C_DIS
LIN {X 0.134,Y -296.607,Z 781.683,A 0.000,B 0.000,C 90.000,E1 302.880} C_DIS
LIN {X 0.006,Y -309.381,Z 781.668,A 0.000,B 0.000,C 90.000,E1 300.256} C_DIS
LIN {X -0.104,Y -327.052,Z 781.650,A 0.000,B 0.000,C 90.000,E1 297.052} C_DIS
LIN {X 0.065,Y -342.333,Z 781.636,A 0.000,B 0.000,C 90.000,E1 294.515} C_DIS
LIN {X 0.141,Y -363.209,Z 781.619,A 0.000,B 0.000,C 90.000,E1 291.461} C_DIS
LIN {X 0.002,Y -384.028,Z 781.605,A 0.000,B 0.000,C 90.000,E1 288.852} C_DIS
LIN {X -0.084,Y -398.989,Z 781.595,A 0.000,B 0.000,C 90.000,E1 287.149} C_DIS
LIN {X -0.159,Y -414.006,Z 781.586,A 0.000,B 0.000,C 90.000,E1 285.481} C_DIS
LIN {X 0.213,Y -426.245,Z 781.578,A 0.000,B 0.000,C 90.000,E1 284.064} C_DIS
LIN {X -0.184,Y -438.092,Z 781.571,A 0.000,B 0.000,C 90.000,E1 282.771} C_DIS
LIN {X -0.208,Y -447.272,Z 781.565,A 0.000,B 0.000,C 90.000,E1 281.715} C_DIS
LIN {X -0.128,Y -455.916,Z 781.559,A 0.000,B 0.000,C 90.000,E1 280.658} C_DIS
LIN {X -0.197,Y -465.788,Z 781.552,A 0.000,B 0.000,C 90.000,E1 279.378} C_DIS
LIN {X -0.051,Y -473.158,Z 781.546,A 0.000,B 0.000,C 90.000,E1 278.341} C_DIS
LIN {X -0.082,Y -478.155,Z 781.542,A 0.000,B 0.000,C 90.000,E1 277.587} C_DIS
LIN {X -0.068,Y -482.519,Z 781.538,A 0.000,B 0.000,C 90.000,E1 276.834} C_DIS
LIN {X -0.076,Y -486.141,Z 781.534,A 0.000,B 0.000,C 90.000,E1 276.087} C_DIS
LIN {X 0.119,Y -488.156,Z 781.531,A 0.000,B 0.000,C 90.000,E1 275.568} C_DIS
LIN {X -0.167,Y -489.796,Z 781.528,A 0.000,B 0.000,C 90.000,E1 275.106} C_DIS
LIN {X 0.044,Y -491.057,Z 781.526,A 0.000,B 0.000,C 90.000,E1 274.588} C_DIS
LIN {X 0.227,Y -491.967,Z 781.523,A 0.000,B 0.000,C 90.000,E1 274.073} C_DIS
LIN {X -0.037,Y -492.450,Z 781.520,A 0.000,B 0.000,C 90.000,E1 273.612} C_DIS
LIN {X 0.192,Y -492.545,Z 781.517,A 0.000,B 0.000,C 90.000,E1 273.094} C_DIS
LIN {X -0.096,Y -492.202,Z 781.515,A 0.000,B 0.000,C 90.000,E1 272.636} C_DIS
LIN {X 0.113,Y -491.452,Z 781.512,A 0.000,B 0.000,C 90.000,E1 272.121} C_DIS
LIN {X -0.156,Y -490.242,Z 781.509,A 0.000,B 0.000,C 90.000,E1 271.661} C_DIS
LIN {X 0.046,Y -488.584,Z 781.506,A 0.000,B 0.000,C 90.000,E1 271.146} C_DIS
LIN {X 0.241,Y -486.490,Z 781.504,A 0.000,B 0.000,C 90.000,E1 270.630} C_DIS
LIN {X -0.059,Y -483.827,Z 781.501,A 0.000,B 0.000,C 90.000,E1 270.172} C_DIS
LIN {X 0.106,Y -480.578,Z 781.498,A 0.000,B 0.000,C 90.000,E1 269.656} C_DIS
LIN {X -0.223,Y -476.518,Z 781.495,A 0.000,B 0.000,C 90.000,E1 269.198} C_DIS
LIN {X 0.078,Y -474.281,Z 781.494,A 0.000,B 0.000,C 90.000,E1 268.912} C_DIS
LIN {X -0.164,Y -468.975,Z 781.491,A 0.000,B 0.000,C 90.000,E1 268.453} C_DIS
LIN {X -0.232,Y -465.939,Z 781.490,A 0.000,B 0.000,C 90.000,E1 268.224} C_DIS
LIN {X 0.079,Y -459.451,Z 781.488,A 0.000,B 0.000,C 90.000,E1 267.764} C_DIS
LIN {X 0.044,Y -456.199,Z 781.487,A 0.000,B 0.000,C 90.000,E1 267.593} C_DIS
LIN {X -0.194,Y -449.007,Z 781.485,A 0.000,B 0.000,C 90.000,E1 267.306} C_DIS
LIN {X 0.096,Y -441.420,Z 781.484,A 0.000,B 0.000,C 90.000,E1 267.020} C_DIS
LIN {X 0.139,Y -437.039,Z 781.483,A 0.000,B 0.000,C 90.000,E1 266.906} C_DIS
LIN {X -0.149,Y -427.197,Z 781.482,A 0.000,B 0.000,C 90.000,E1 266.788} C_DIS
LIN {X -0.115,Y -418.313,Z 781.482,A 0.000,B 0.000,C 90.000,E1 266.731} C_DIS
LIN {X -0.068,Y -180.964,Z 781.482,A 0.000,B 0.000,C 90.000,E1 266.731} C_DIS
LIN {X -0.062,Y -180.859,Z 781.472,A 0.000,B 0.000,C 90.000,E1 265.008} C_DIS
LIN {X -0.008,Y -178.972,Z 781.444,A 0.000,B 0.000,C 90.000,E1 259.926} C_DIS
LIN {X 0.002,Y -177.930,Z 781.435,A 0.000,B 0.000,C 90.000,E1 258.229} C_DIS
LIN {X 0.017,Y -175.569,Z 781.411,A 0.000,B 0.000,C 90.000,E1 253.976} C_DIS
LIN {X 0.024,Y -172.297,Z 781.387,A 0.000,B 0.000,C 90.000,E1 249.699} C_DIS
LIN {X 0.001,Y -171.775,Z 781.383,A 0.000,B 0.000,C 90.000,E1 248.847} C_DIS
LIN {X -0.026,Y -168.704,Z 781.363,A 0.000,B 0.000,C 90.000,E1 245.409} C_DIS
LIN {X 0.013,Y -166.769,Z 781.349,A 0.000,B 0.000,C 90.000,E1 242.794} C_DIS
LIN {X 0.071,Y -162.749,Z 781.325,A 0.000,B 0.000,C 90.000,E1 238.408} C_DIS
LIN {X -0.091,Y -161.439,Z 781.315,A 0.000,B 0.000,C 90.000,E1 236.707} C_DIS
LIN {X -0.049,Y -157.432,Z 781.290,A 0.000,B 0.000,C 90.000,E1 232.271} C_DIS
LIN {X -0.014,Y -155.438,Z 781.275,A 0.000,B 0.000,C 90.000,E1 229.585} C_DIS
LIN {X 0.034,Y -151.759,Z 781.251,A 0.000,B 0.000,C 90.000,E1 225.081} C_DIS
LIN {X 0.046,Y -149.960,Z 781.235,A 0.000,B 0.000,C 90.000,E1 222.366} C_DIS
LIN {X 0.073,Y -146.802,Z 781.210,A 0.000,B 0.000,C 90.000,E1 217.810} C_DIS
LIN {X -0.027,Y -145.377,Z 781.195,A 0.000,B 0.000,C 90.000,E1 215.105} C_DIS
LIN {X -0.034,Y -142.439,Z 781.164,A 0.000,B 0.000,C 90.000,E1 209.589} C_DIS
LIN {X 0.013,Y -141.429,Z 781.149,A 0.000,B 0.000,C 90.000,E1 206.796} C_DIS
LIN {X -0.006,Y -139.365,Z 781.113,A 0.000,B 0.000,C 90.000,E1 200.301} C_DIS
LIN {X -0.020,Y -138.810,Z 781.097,A 0.000,B 0.000,C 90.000,E1 197.511} C_DIS
LIN {X 0.030,Y -138.351,Z 781.056,A 0.000,B 0.000,C 90.000,E1 190.018} C_DIS
LIN {X 0.007,Y -139.541,Z 781.004,A 0.000,B 0.000,C 90.000,E1 180.688} C_DIS
LIN {X -0.041,Y -141.237,Z 780.973,A 0.000,B 0.000,C 90.000,E1 175.122} C_DIS
LIN {X 0.059,Y -142.608,Z 780.957,A 0.000,B 0.000,C 90.000,E1 172.299} C_DIS
LIN {X 0.012,Y -144.919,Z 780.932,A 0.000,B 0.000,C 90.000,E1 167.701} C_DIS
LIN {X 0.004,Y -147.548,Z 780.911,A 0.000,B 0.000,C 90.000,E1 164.031} C_DIS
LIN {X 0.036,Y -150.151,Z 780.891,A 0.000,B 0.000,C 90.000,E1 160.369} C_DIS
LIN {X 0.046,Y -153.520,Z 780.871,A 0.000,B 0.000,C 90.000,E1 156.741} C_DIS
LIN {X -0.033,Y -157.886,Z 780.846,A 0.000,B 0.000,C 90.000,E1 152.281} C_DIS
LIN {X -0.079,Y -162.173,Z 780.826,A 0.000,B 0.000,C 90.000,E1 148.742} C_DIS
LIN {X 0.035,Y -166.382,Z 780.807,A 0.000,B 0.000,C 90.000,E1 145.182} C_DIS
LIN {X 0.039,Y -171.398,Z 780.787,A 0.000,B 0.000,C 90.000,E1 141.698} C_DIS
LIN {X 0.078,Y -176.311,Z 780.768,A 0.000,B 0.000,C 90.000,E1 138.243} C_DIS
LIN {X -0.054,Y -180.598,Z 780.754,A 0.000,B 0.000,C 90.000,E1 135.729} C_DIS
LIN {X -0.076,Y -186.000,Z 780.735,A 0.000,B 0.000,C 90.000,E1 132.366} C_DIS
LIN {X -0.021,Y -190.634,Z 780.721,A 0.000,B 0.000,C 90.000,E1 129.850} C_DIS
LIN {X -0.024,Y -192.467,Z 780.715,A 0.000,B 0.000,C 90.000,E1 128.749} C_DIS
LIN {X -0.072,Y -292.357,Z 780.715,A 0.000,B 0.000,C 90.000,E1 128.749} C_DIS
LIN {X 0.044,Y -294.992,Z 780.715,A 0.000,B 0.000,C 90.000,E1 128.669} C_DIS
LIN {X -0.150,Y -299.262,Z 780.714,A 0.000,B 0.000,C 90.000,E1 128.463} C_DIS
LIN {X 0.077,Y -301.787,Z 780.712,A 0.000,B 0.000,C 90.000,E1 128.177} C_DIS
LIN {X -0.040,Y -305.547,Z 780.709,A 0.000,B 0.000,C 90.000,E1 127.649} C_DIS
LIN {X -0.029,Y -307.116,Z 780.707,A 0.000,B 0.000,C 90.000,E1 127.317} C_DIS
LIN {X -0.076,Y -308.350,Z 780.705,A 0.000,B 0.000,C 90.000,E1 126.996} C_DIS
LIN {X -0.032,Y -319.314,Z 780.686,A 0.000,B 0.000,C 90.000,E1 123.420} C_DIS
LIN {X 0.054,Y -329.623,Z 780.670,A 0.000,B 0.000,C 90.000,E1 120.541} C_DIS
LIN {X 0.124,Y -341.273,Z 780.654,A 0.000,B 0.000,C 90.000,E1 117.719} C_DIS
LIN {X 0.053,Y -354.374,Z 780.639,A 0.000,B 0.000,C 90.000,E1 114.975} C_DIS
LIN {X -0.019,Y -367.329,Z 780.625,A 0.000,B 0.000,C 90.000,E1 112.589} C_DIS
LIN {X -0.057,Y -381.613,Z 780.612,A 0.000,B 0.000,C 90.000,E1 110.248} C_DIS
LIN {X 0.002,Y -397.330,Z 780.600,A 0.000,B 0.000,C 90.000,E1 107.946} C_DIS
LIN {X -0.061,Y -414.591,Z 780.587,A 0.000,B 0.000,C 90.000,E1 105.717} C_DIS
LIN {X -0.040,Y -433.523,Z 780.575,A 0.000,B 0.000,C 90.000,E1 103.536} C_DIS
LIN {X 0.004,Y -453.585,Z 780.564,A 0.000,B 0.000,C 90.000,E1 101.478} C_DIS
LIN {X -0.178,Y -468.801,Z 780.556,A 0.000,B 0.000,C 90.000,E1 100.074} C_DIS
LIN {X 0.146,Y -470.695,Z 780.555,A 0.000,B 0.000,C 90.000,E1 99.792} C_DIS
LIN {X 0.088,Y -472.132,Z 780.553,A 0.000,B 0.000,C 90.000,E1 99.557} C_DIS
LIN {X 0.265,Y -474.072,Z 780.550,A 0.000,B 0.000,C 90.000,E1 99.029} C_DIS
LIN {X -0.092,Y -474.897,Z 780.548,A 0.000,B 0.000,C 90.000,E1 98.568} C_DIS
LIN {X 0.033,Y -474.748,Z 780.545,A 0.000,B 0.000,C 90.000,E1 98.049} C_DIS
LIN {X 0.164,Y -473.606,Z 780.542,A 0.000,B 0.000,C 90.000,E1 97.530} C_DIS
LIN {X 0.024,Y -472.611,Z 780.541,A 0.000,B 0.000,C 90.000,E1 97.296} C_DIS
LIN {X -0.174,Y -471.272,Z 780.539,A 0.000,B 0.000,C 90.000,E1 97.068} C_DIS
LIN {X -0.006,Y -453.491,Z 780.524,A 0.000,B 0.000,C 90.000,E1 94.245} C_DIS
LIN {X 0.136,Y -442.939,Z 780.513,A 0.000,B 0.000,C 90.000,E1 92.407} C_DIS
LIN {X -0.120,Y -433.811,Z 780.505,A 0.000,B 0.000,C 90.000,E1 90.859} C_DIS
LIN {X -0.106,Y -424.356,Z 780.496,A 0.000,B 0.000,C 90.000,E1 89.255} C_DIS
LIN {X -0.154,Y -413.122,Z 780.485,A 0.000,B 0.000,C 90.000,E1 87.364} C_DIS
LIN {X -0.057,Y -403.402,Z 780.476,A 0.000,B 0.000,C 90.000,E1 85.698} C_DIS
LIN {X -0.020,Y -390.358,Z 780.464,A 0.000,B 0.000,C 90.000,E1 83.451} C_DIS
LIN {X 0.154,Y -376.163,Z 780.449,A 0.000,B 0.000,C 90.000,E1 80.849} C_DIS
LIN {X 0.028,Y -360.905,Z 780.433,A 0.000,B 0.000,C 90.000,E1 77.937} C_DIS
LIN {X 0.163,Y -349.380,Z 780.420,A 0.000,B 0.000,C 90.000,E1 75.519} C_DIS
LIN {X 0.099,Y -337.884,Z 780.406,A 0.000,B 0.000,C 90.000,E1 73.087} C_DIS
LIN {X 0.056,Y -326.683,Z 780.392,A 0.000,B 0.000,C 90.000,E1 70.604} C_DIS
LIN {X 0.132,Y -313.166,Z 780.375,A 0.000,B 0.000,C 90.000,E1 67.411} C_DIS
LIN {X 0.034,Y -299.360,Z 780.355,A 0.000,B 0.000,C 90.000,E1 63.845} C_DIS
LIN {X -0.123,Y -286.878,Z 780.334,A 0.000,B 0.000,C 90.000,E1 60.205} C_DIS
LIN {X -0.046,Y -276.372,Z 780.315,A 0.000,B 0.000,C 90.000,E1 56.786} C_DIS
LIN {X 0.080,Y -268.238,Z 780.300,A 0.000,B 0.000,C 90.000,E1 53.989} C_DIS
LIN {X -0.015,Y -262.190,Z 780.288,A 0.000,B 0.000,C 90.000,E1 51.904} C_DIS
LIN {X -0.011,Y -254.200,Z 780.273,A 0.000,B 0.000,C 90.000,E1 49.057} C_DIS
LIN {X 0.119,Y -244.500,Z 780.252,A 0.000,B 0.000,C 90.000,E1 45.405} C_DIS
LIN {X 0.001,Y -237.049,Z 780.236,A 0.000,B 0.000,C 90.000,E1 42.486} C_DIS
LIN {X -0.040,Y -227.994,Z 780.215,A 0.000,B 0.000,C 90.000,E1 38.749} C_DIS
LIN {X 0.092,Y -219.443,Z 780.194,A 0.000,B 0.000,C 90.000,E1 34.898} C_DIS
LIN {X -0.055,Y -211.618,Z 780.172,A 0.000,B 0.000,C 90.000,E1 31.052} C_DIS
LIN {X -0.051,Y -206.037,Z 780.155,A 0.000,B 0.000,C 90.000,E1 27.897} C_DIS
LIN {X -0.037,Y -200.190,Z 780.133,A 0.000,B 0.000,C 90.000,E1 23.898} C_DIS
LIN {X 0.108,Y -195.407,Z 780.110,A 0.000,B 0.000,C 90.000,E1 19.812} C_DIS
LIN {X -0.102,Y -191.728,Z 780.088,A 0.000,B 0.000,C 90.000,E1 15.788} C_DIS
LIN {X -0.081,Y -188.733,Z 780.060,A 0.000,B 0.000,C 90.000,E1 10.838} C_DIS
LIN {X 0.061,Y -187.829,Z 779.984,A 0.000,B 0.000,C 90.000,E1 357.020} C_DIS
LIN {X -0.048,Y -190.574,Z 779.951,A 0.000,B 0.000,C 90.000,E1 351.254} C_DIS
LIN {X 0.014,Y -194.333,Z 779.924,A 0.000,B 0.000,C 90.000,E1 346.297} C_DIS
LIN {X -0.054,Y -198.543,Z 779.901,A 0.000,B 0.000,C 90.000,E1 342.236} C_DIS
LIN {X 0.081,Y -203.882,Z 779.879,A 0.000,B 0.000,C 90.000,E1 338.156} C_DIS
LIN {X -0.065,Y -210.123,Z 779.857,A 0.000,B 0.000,C 90.000,E1 334.204} C_DIS
LIN {X -0.026,Y -217.253,Z 779.835,A 0.000,B 0.000,C 90.000,E1 330.255} C_DIS
LIN {X -0.008,Y -225.078,Z 779.813,A 0.000,B 0.000,C 90.000,E1 326.373} C_DIS
LIN {X 0.005,Y -233.589,Z 779.792,A 0.000,B 0.000,C 90.000,E1 322.557} C_DIS
LIN {X 0.018,Y -242.869,Z 779.771,A 0.000,B 0.000,C 90.000,E1 318.809} C_DIS
LIN {X 0.084,Y -251.961,Z 779.753,A 0.000,B 0.000,C 90.000,E1 315.486} C_DIS
LIN {X -0.064,Y -262.801,Z 779.733,A 0.000,B 0.000,C 90.000,E1 311.919} C_DIS
LIN {X -0.089,Y -273.513,Z 779.715,A 0.000,B 0.000,C 90.000,E1 308.749} C_DIS
LIN {X 0.123,Y -285.229,Z 779.698,A 0.000,B 0.000,C 90.000,E1 305.598} C_DIS
LIN {X -0.063,Y -298.056,Z 779.681,A 0.000,B 0.000,C 90.000,E1 302.594} C_DIS
LIN {X 0.100,Y -311.037,Z 779.666,A 0.000,B 0.000,C 90.000,E1 299.922} C_DIS
LIN {X -0.102,Y -328.853,Z 779.648,A 0.000,B 0.000,C 90.000,E1 296.744} C_DIS
LIN {X 0.126,Y -342.259,Z 779.636,A 0.000,B 0.000,C 90.000,E1 294.515} C_DIS
LIN {X 0.070,Y -363.080,Z 779.619,A 0.000,B 0.000,C 90.000,E1 291.482} C_DIS
LIN {X -0.057,Y -383.962,Z 779.605,A 0.000,B 0.000,C 90.000,E1 288.852} C_DIS
LIN {X -0.090,Y -398.858,Z 779.595,A 0.000,B 0.000,C 90.000,E1 287.149} C_DIS
LIN {X -0.093,Y -413.741,Z 779.586,A 0.000,B 0.000,C 90.000,E1 285.481} C_DIS
LIN {X -0.131,Y -425.952,Z 779.578,A 0.000,B 0.000,C 90.000,E1 284.120} C_DIS
LIN {X -0.118,Y -437.778,Z 779.571,A 0.000,B 0.000,C 90.000,E1 282.771} C_DIS
LIN {X 0.089,Y -449.159,Z 779.564,A 0.000,B 0.000,C 90.000,E1 281.422} C_DIS
LIN {X 0.196,Y -457.609,Z 779.558,A 0.000,B 0.000,C 90.000,E1 280.366} C_DIS
LIN {X 0.077,Y -467.385,Z 779.551,A 0.000,B 0.000,C 90.000,E1 279.095} C_DIS
LIN {X 0.003,Y -472.893,Z 779.546,A 0.000,B 0.000,C 90.000,E1 278.341} C_DIS
LIN {X -0.030,Y -477.923,Z 779.542,A 0.000,B 0.000,C 90.000,E1 277.587} C_DIS
LIN {X -0.017,Y -482.345,Z 779.538,A 0.000,B 0.000,C 90.000,E1 276.834} C_DIS
LIN {X -0.026,Y -486.019,Z 779.534,A 0.000,B 0.000,C 90.000,E1 276.087} C_DIS
LIN {X 0.168,Y -488.047,Z 779.531,A 0.000,B 0.000,C 90.000,E1 275.568} C_DIS
LIN {X -0.118,Y -489.721,Z 779.528,A 0.000,B 0.000,C 90.000,E1 275.106} C_DIS
LIN {X 0.092,Y -491.007,Z 779.526,A 0.000,B 0.000,C 90.000,E1 274.588} C_DIS
LIN {X -0.215,Y -491.949,Z 779.523,A 0.000,B 0.000,C 90.000,E1 274.131} C_DIS
LIN {X 0.011,Y -492.453,Z 779.520,A 0.000,B 0.000,C 90.000,E1 273.612} C_DIS
LIN {X 0.240,Y -492.586,Z 779.517,A 0.000,B 0.000,C 90.000,E1 273.094} C_DIS
LIN {X -0.048,Y -492.264,Z 779.515,A 0.000,B 0.000,C 90.000,E1 272.636} C_DIS
LIN {X 0.160,Y -491.554,Z 779.512,A 0.000,B 0.000,C 90.000,E1 272.121} C_DIS
LIN {X -0.108,Y -490.396,Z 779.509,A 0.000,B 0.000,C 90.000,E1 271.661} C_DIS
LIN {X 0.095,Y -488.773,Z 779.506,A 0.000,B 0.000,C 90.000,E1 271.146} C_DIS
LIN {X -0.197,Y -486.664,Z 779.504,A 0.000,B 0.000,C 90.000,E1 270.688} C_DIS
LIN {X -0.009,Y -484.015,Z 779.501,A 0.000,B 0.000,C 90.000,E1 270.172} C_DIS
LIN {X 0.158,Y -480.764,Z 779.498,A 0.000,B 0.000,C 90.000,E1 269.656} C_DIS
LIN {X -0.172,Y -476.755,Z 779.495,A 0.000,B 0.000,C 90.000,E1 269.198} C_DIS
LIN {X 0.130,Y -474.488,Z 779.494,A 0.000,B 0.000,C 90.000,E1 268.912} C_DIS
LIN {X -0.141,Y -469.161,Z 779.491,A 0.000,B 0.000,C 90.000,E1 268.453} C_DIS
LIN {X -0.236,Y -466.116,Z 779.490,A 0.000,B 0.000,C 90.000,E1 268.224} C_DIS
LIN {X 0.047,Y -459.656,Z 779.488,A 0.000,B 0.000,C 90.000,E1 267.764} C_DIS
LIN {X -0.007,Y -456.379,Z 779.487,A 0.000,B 0.000,C 90.000,E1 267.593} C_DIS
LIN {X 0.185,Y -449.153,Z 779.485,A 0.000,B 0.000,C 90.000,E1 267.249} C_DIS
LIN {X 0.034,Y -441.608,Z 779.483,A 0.000,B 0.000,C 90.000,E1 267.020} C_DIS
LIN {X 0.084,Y -437.285,Z 779.483,A 0.000,B 0.000,C 90.000,E1 266.906} C_DIS
LIN {X 0.218,Y -427.576,Z 779.482,A 0.000,B 0.000,C 90.000,E1 266.731} C_DIS
LIN {X -0.117,Y -422.213,Z 779.482,A 0.000,B 0.000,C 90.000,E1 266.731} C_DIS
LIN {X 0.205,Y -415.673,Z 779.482,A 0.000,B 0.000,C 90.000,E1 266.674} C_DIS
LIN {X 0.068,Y -180.964,Z 779.482,A 0.000,B 0.000,C 90.000,E1 266.674} C_DIS
LIN {X 0.084,Y -180.856,Z 779.472,A 0.000,B 0.000,C 90.000,E1 264.951} C_DIS
LIN {X -0.043,Y -178.968,Z 779.444,A 0.000,B 0.000,C 90.000,E1 259.926} C_DIS
LIN {X -0.032,Y -177.923,Z 779.435,A 0.000,B 0.000,C 90.000,E1 258.229} C_DIS
LIN {X -0.017,Y -175.560,Z 779.411,A 0.000,B 0.000,C 90.000,E1 253.976} C_DIS
LIN {X -0.010,Y -172.290,Z 779.387,A 0.000,B 0.000,C 90.000,E1 249.699} C_DIS
LIN {X -0.032,Y -171.769,Z 779.382,A 0.000,B 0.000,C 90.000,E1 248.847} C_DIS
LIN {X -0.040,Y -168.010,Z 779.358,A 0.000,B 0.000,C 90.000,E1 244.537} C_DIS
LIN {X -0.020,Y -166.760,Z 779.349,A 0.000,B 0.000,C 90.000,E1 242.794} C_DIS
LIN {X 0.039,Y -162.739,Z 779.325,A 0.000,B 0.000,C 90.000,E1 238.408} C_DIS
LIN {X 0.100,Y -161.430,Z 779.315,A 0.000,B 0.000,C 90.000,E1 236.628} C_DIS
LIN {X -0.080,Y -157.424,Z 779.290,A 0.000,B 0.000,C 90.000,E1 232.271} C_DIS
LIN {X 0.072,Y -155.427,Z 779.275,A 0.000,B 0.000,C 90.000,E1 229.542} C_DIS
LIN {X 0.003,Y -151.751,Z 779.250,A 0.000,B 0.000,C 90.000,E1 225.081} C_DIS
LIN {X 0.015,Y -149.951,Z 779.235,A 0.000,B 0.000,C 90.000,E1 222.366} C_DIS
LIN {X 0.042,Y -146.794,Z 779.210,A 0.000,B 0.000,C 90.000,E1 217.810} C_DIS
LIN {X -0.057,Y -145.369,Z 779.195,A 0.000,B 0.000,C 90.000,E1 215.105} C_DIS
LIN {X 0.059,Y -142.433,Z 779.164,A 0.000,B 0.000,C 90.000,E1 209.539} C_DIS
LIN {X -0.018,Y -141.424,Z 779.149,A 0.000,B 0.000,C 90.000,E1 206.796} C_DIS
LIN {X -0.036,Y -139.363,Z 779.113,A 0.000,B 0.000,C 90.000,E1 200.301} C_DIS
LIN {X -0.049,Y -138.808,Z 779.097,A 0.000,B 0.000,C 90.000,E1 197.511} C_DIS
LIN {X 0.001,Y -138.351,Z 779.056,A 0.000,B 0.000,C 90.000,E1 190.018} C_DIS
LIN {X -0.023,Y -139.543,Z 779.004,A 0.000,B 0.000,C 90.000,E1 180.688} C_DIS
LIN {X 0.070,Y -141.243,Z 778.973,A 0.000,B 0.000,C 90.000,E1 175.065} C_DIS
LIN {X 0.029,Y -142.612,Z 778.957,A 0.000,B 0.000,C 90.000,E1 172.299} C_DIS
LIN {X -0.018,Y -144.927,Z 778.932,A 0.000,B 0.000,C 90.000,E1 167.701} C_DIS
LIN {X -0.027,Y -147.555,Z 778.911,A 0.000,B 0.000,C 90.000,E1 164.031} C_DIS
LIN {X 0.005,Y -150.160,Z 778.891,A 0.000,B 0.000,C 90.000,E1 160.369} C_DIS
LIN {X 0.015,Y -153.533,Z 778.871,A 0.000,B 0.000,C 90.000,E1 156.741} C_DIS
LIN {X 0.067,Y -156.950,Z 778.851,A 0.000,B 0.000,C 90.000,E1 153.127} C_DIS
LIN {X 0.003,Y -161.055,Z 778.831,A 0.000,B 0.000,C 90.000,E1 149.587} C_DIS
LIN {X 0.087,Y -163.164,Z 778.821,A 0.000,B 0.000,C 90.000,E1 147.788} C_DIS
LIN {X -0.042,Y -167.583,Z 778.802,A 0.000,B 0.000,C 90.000,E1 144.322} C_DIS
LIN {X 0.004,Y -171.412,Z 778.787,A 0.000,B 0.000,C 90.000,E1 141.698} C_DIS
LIN {X 0.043,Y -176.328,Z 778.768,A 0.000,B 0.000,C 90.000,E1 138.243} C_DIS
LIN {X -0.089,Y -180.617,Z 778.754,A 0.000,B 0.000,C 90.000,E1 135.729} C_DIS
LIN {X 0.026,Y -186.019,Z 778.735,A 0.000,B 0.000,C 90.000,E1 132.324} C_DIS
LIN {X -0.057,Y -190.654,Z 778.721,A 0.000,B 0.000,C 90.000,E1 129.850} C_DIS
LIN {X 0.037,Y -192.437,Z 778.715,A 0.000,B 0.000,C 90.000,E1 128.749} C_DIS
LIN {X 0.007,Y -291.854,Z 778.715,A 0.000,B 0.000,C 90.000,E1 128.749} C_DIS
LIN {X -0.091,Y -293.401,Z 778.715,A 0.000,B 0.000,C 90.000,E1 128.749} C_DIS
LIN {X -0.037,Y -299.091,Z 778.714,A 0.000,B 0.000,C 90.000,E1 128.463} C_DIS
LIN {X 0.021,Y -301.935,Z 778.712,A 0.000,B 0.000,C 90.000,E1 128.177} C_DIS
LIN {X -0.113,Y -305.631,Z 778.709,A 0.000,B 0.000,C 90.000,E1 127.649} C_DIS
LIN {X -0.102,Y -307.170,Z 778.707,A 0.000,B 0.000,C 90.000,E1 127.317} C_DIS
LIN {X 0.098,Y -308.379,Z 778.705,A 0.000,B 0.000,C 90.000,E1 126.950} C_DIS
LIN {X 0.160,Y -319.338,Z 778.686,A 0.000,B 0.000,C 90.000,E1 123.372} C_DIS
LIN {X -0.021,Y -329.651,Z 778.670,A 0.000,B 0.000,C 90.000,E1 120.541} C_DIS
LIN {X 0.046,Y -341.308,Z 778.654,A 0.000,B 0.000,C 90.000,E1 117.719} C_DIS
LIN {X 0.124,Y -354.417,Z 778.639,A 0.000,B 0.000,C 90.000,E1 114.951} C_DIS
LIN {X -0.100,Y -367.377,Z 778.625,A 0.000,B 0.000,C 90.000,E1 112.589} C_DIS
LIN {X -0.139,Y -381.669,Z 778.612,A 0.000,B 0.000,C 90.000,E1 110.248} C_DIS
LIN {X -0.083,Y -397.393,Z 778.600,A 0.000,B 0.000,C 90.000,E1 107.946} C_DIS
LIN {X -0.147,Y -414.662,Z 778.587,A 0.000,B 0.000,C 90.000,E1 105.717} C_DIS
LIN {X -0.129,Y -433.604,Z 778.575,A 0.000,B 0.000,C 90.000,E1 103.536} C_DIS
LIN {X -0.083,Y -453.668,Z 778.564,A 0.000,B 0.000,C 90.000,E1 101.478} C_DIS
LIN {X 0.172,Y -466.479,Z 778.557,A 0.000,B 0.000,C 90.000,E1 100.254} C_DIS
LIN {X 0.199,Y -468.872,Z 778.556,A 0.000,B 0.000,C 90.000,E1 100.018} C_DIS
LIN {X 0.053,Y -470.756,Z 778.554,A 0.000,B 0.000,C 90.000,E1 99.792} C_DIS
LIN {X -0.012,Y -472.186,Z 778.553,A 0.000,B 0.000,C 90.000,E1 99.557} C_DIS
LIN {X 0.166,Y -474.105,Z 778.550,A 0.000,B 0.000,C 90.000,E1 99.029} C_DIS
LIN {X -0.192,Y -474.912,Z 778.547,A 0.000,B 0.000,C 90.000,E1 98.568} C_DIS
LIN {X -0.067,Y -474.747,Z 778.545,A 0.000,B 0.000,C 90.000,E1 98.049} C_DIS
LIN {X 0.064,Y -473.588,Z 778.542,A 0.000,B 0.000,C 90.000,E1 97.530} C_DIS
LIN {X -0.075,Y -472.582,Z 778.540,A 0.000,B 0.000,C 90.000,E1 97.296} C_DIS
LIN {X 0.195,Y -471.230,Z 778.539,A 0.000,B 0.000,C 90.000,E1 97.011} C_DIS
LIN {X -0.102,Y -453.449,Z 778.523,A 0.000,B 0.000,C 90.000,E1 94.245} C_DIS
LIN {X 0.040,Y -442.897,Z 778.513,A 0.000,B 0.000,C 90.000,E1 92.407} C_DIS
LIN {X -0.214,Y -433.779,Z 778.505,A 0.000,B 0.000,C 90.000,E1 90.859} C_DIS
LIN {X -0.198,Y -424.335,Z 778.496,A 0.000,B 0.000,C 90.000,E1 89.255} C_DIS
LIN {X 0.169,Y -413.111,Z 778.485,A 0.000,B 0.000,C 90.000,E1 87.306} C_DIS
LIN {X -0.147,Y -403.391,Z 778.476,A 0.000,B 0.000,C 90.000,E1 85.698} C_DIS
LIN {X -0.106,Y -390.355,Z 778.464,A 0.000,B 0.000,C 90.000,E1 83.451} C_DIS
LIN {X 0.084,Y -374.624,Z 778.448,A 0.000,B 0.000,C 90.000,E1 80.557} C_DIS
LIN {X -0.117,Y -358.023,Z 778.430,A 0.000,B 0.000,C 90.000,E1 77.353} C_DIS
LIN {X 0.018,Y -347.957,Z 778.418,A 0.000,B 0.000,C 90.000,E1 75.227} C_DIS
LIN {X -0.090,Y -335.110,Z 778.403,A 0.000,B 0.000,C 90.000,E1 72.489} C_DIS
LIN {X -0.197,Y -323.981,Z 778.389,A 0.000,B 0.000,C 90.000,E1 70.007} C_DIS
LIN {X -0.084,Y -310.664,Z 778.371,A 0.000,B 0.000,C 90.000,E1 66.794} C_DIS
LIN {X 0.004,Y -297.163,Z 778.351,A 0.000,B 0.000,C 90.000,E1 63.179} C_DIS
LIN {X -0.173,Y -287.091,Z 778.334,A 0.000,B 0.000,C 90.000,E1 60.205} C_DIS
LIN {X 0.071,Y -276.644,Z 778.315,A 0.000,B 0.000,C 90.000,E1 56.755} C_DIS
LIN {X 0.054,Y -268.557,Z 778.300,A 0.000,B 0.000,C 90.000,E1 53.989} C_DIS
LIN {X -0.035,Y -262.545,Z 778.288,A 0.000,B 0.000,C 90.000,E1 51.904} C_DIS
LIN {X -0.022,Y -254.572,Z 778.273,A 0.000,B 0.000,C 90.000,E1 49.057} C_DIS
LIN {X 0.122,Y -246.780,Z 778.256,A 0.000,B 0.000,C 90.000,E1 46.134} C_DIS
LIN {X 0.085,Y -241.168,Z 778.244,A 0.000,B 0.000,C 90.000,E1 43.947} C_DIS
LIN {X 0.053,Y -233.731,Z 778.228,A 0.000,B 0.000,C 90.000,E1 40.987} C_DIS
LIN {X 0.067,Y -226.600,Z 778.211,A 0.000,B 0.000,C 90.000,E1 37.971} C_DIS
LIN {X -0.149,Y -218.155,Z 778.190,A 0.000,B 0.000,C 90.000,E1 34.199} C_DIS
LIN {X 0.030,Y -210.472,Z 778.168,A 0.000,B 0.000,C 90.000,E1 30.256} C_DIS
LIN {X -0.095,Y -205.077,Z 778.151,A 0.000,B 0.000,C 90.000,E1 27.129} C_DIS
LIN {X 0.074,Y -199.430,Z 778.128,A 0.000,B 0.000,C 90.000,E1 23.078} C_DIS
LIN {X 0.051,Y -194.866,Z 778.106,A 0.000,B 0.000,C 90.000,E1 19.033} C_DIS
LIN {X 0.014,Y -191.348,Z 778.083,A 0.000,B 0.000,C 90.000,E1 14.954} C_DIS
LIN {X -0.085,Y -188.282,Z 778.051,A 0.000,B 0.000,C 90.000,E1 9.208} C_DIS
LIN {X 0.064,Y -187.966,Z 777.984,A 0.000,B 0.000,C 90.000,E1 357.020} C_DIS
LIN {X -0.039,Y -190.697,Z 777.951,A 0.000,B 0.000,C 90.000,E1 351.254} C_DIS
LIN {X 0.028,Y -194.473,Z 777.924,A 0.000,B 0.000,C 90.000,E1 346.297} C_DIS
LIN {X -0.035,Y -198.688,Z 777.901,A 0.000,B 0.000,C 90.000,E1 342.236} C_DIS
LIN {X 0.105,Y -204.021,Z 777.879,A 0.000,B 0.000,C 90.000,E1 338.156} C_DIS
LIN {X -0.037,Y -210.258,Z 777.857,A 0.000,B 0.000,C 90.000,E1 334.204} C_DIS
LIN {X 0.009,Y -217.380,Z 777.835,A 0.000,B 0.000,C 90.000,E1 330.255} C_DIS
LIN {X 0.031,Y -225.197,Z 777.813,A 0.000,B 0.000,C 90.000,E1 326.373} C_DIS
LIN {X 0.050,Y -233.687,Z 777.792,A 0.000,B 0.000,C 90.000,E1 322.557} C_DIS
LIN {X -0.115,Y -242.937,Z 777.771,A 0.000,B 0.000,C 90.000,E1 318.852} C_DIS
LIN {X -0.038,Y -253.048,Z 777.751,A 0.000,B 0.000,C 90.000,E1 315.162} C_DIS
LIN {X 0.040,Y -263.979,Z 777.731,A 0.000,B 0.000,C 90.000,E1 311.553} C_DIS
LIN {X 0.148,Y -276.004,Z 777.711,A 0.000,B 0.000,C 90.000,E1 308.016} C_DIS
LIN {X 0.007,Y -289.328,Z 777.692,A 0.000,B 0.000,C 90.000,E1 304.612} C_DIS
LIN {X 0.005,Y -299.531,Z 777.679,A 0.000,B 0.000,C 90.000,E1 302.260} C_DIS
LIN {X 0.166,Y -316.153,Z 777.661,A 0.000,B 0.000,C 90.000,E1 298.949} C_DIS
LIN {X -0.013,Y -334.373,Z 777.643,A 0.000,B 0.000,C 90.000,E1 295.796} C_DIS
LIN {X -0.126,Y -344.198,Z 777.635,A 0.000,B 0.000,C 90.000,E1 294.259} C_DIS
LIN {X -0.139,Y -365.165,Z 777.618,A 0.000,B 0.000,C 90.000,E1 291.227} C_DIS
LIN {X 0.146,Y -386.186,Z 777.603,A 0.000,B 0.000,C 90.000,E1 288.544} C_DIS
LIN {X 0.028,Y -401.135,Z 777.594,A 0.000,B 0.000,C 90.000,E1 286.858} C_DIS
LIN {X 0.126,Y -415.899,Z 777.584,A 0.000,B 0.000,C 90.000,E1 285.190} C_DIS
LIN {X 0.099,Y -428.051,Z 777.577,A 0.000,B 0.000,C 90.000,E1 283.828} C_DIS
LIN {X 0.183,Y -439.728,Z 777.569,A 0.000,B 0.000,C 90.000,E1 282.479} C_DIS
LIN {X 0.000,Y -450.949,Z 777.562,A 0.000,B 0.000,C 90.000,E1 281.186} C_DIS
LIN {X 0.044,Y -459.221,Z 777.556,A 0.000,B 0.000,C 90.000,E1 280.141} C_DIS
LIN {X 0.191,Y -467.022,Z 777.551,A 0.000,B 0.000,C 90.000,E1 279.095} C_DIS
LIN {X 0.115,Y -472.564,Z 777.546,A 0.000,B 0.000,C 90.000,E1 278.341} C_DIS
LIN {X 0.080,Y -477.687,Z 777.542,A 0.000,B 0.000,C 90.000,E1 277.587} C_DIS
LIN {X 0.092,Y -482.122,Z 777.538,A 0.000,B 0.000,C 90.000,E1 276.834} C_DIS
LIN {X 0.082,Y -485.857,Z 777.534,A 0.000,B 0.000,C 90.000,E1 276.087} C_DIS
LIN {X -0.211,Y -487.916,Z 777.531,A 0.000,B 0.000,C 90.000,E1 275.625} C_DIS
LIN {X -0.005,Y -489.627,Z 777.528,A 0.000,B 0.000,C 90.000,E1 275.106} C_DIS
LIN {X 0.204,Y -490.946,Z 777.526,A 0.000,B 0.000,C 90.000,E1 274.588} C_DIS
LIN {X -0.104,Y -491.905,Z 777.523,A 0.000,B 0.000,C 90.000,E1 274.131} C_DIS
LIN {X 0.123,Y -492.472,Z 777.520,A 0.000,B 0.000,C 90.000,E1 273.612} C_DIS
LIN {X -0.140,Y -492.618,Z 777.517,A 0.000,B 0.000,C 90.000,E1 273.151} C_DIS
LIN {X 0.063,Y -492.347,Z 777.515,A 0.000,B 0.000,C 90.000,E1 272.636} C_DIS
LIN {X -0.219,Y -491.682,Z 777.512,A 0.000,B 0.000,C 90.000,E1 272.178} C_DIS
LIN {X 0.004,Y -490.574,Z 777.509,A 0.000,B 0.000,C 90.000,E1 271.661} C_DIS
LIN {X 0.206,Y -488.985,Z 777.506,A 0.000,B 0.000,C 90.000,E1 271.146} C_DIS
LIN {X -0.084,Y -486.875,Z 777.504,A 0.000,B 0.000,C 90.000,E1 270.688} C_DIS
LIN {X 0.104,Y -484.237,Z 777.501,A 0.000,B 0.000,C 90.000,E1 270.172} C_DIS
LIN {X -0.210,Y -481.013,Z 777.498,A 0.000,B 0.000,C 90.000,E1 269.714} C_DIS
LIN {X -0.057,Y -477.084,Z 777.495,A 0.000,B 0.000,C 90.000,E1 269.198} C_DIS
LIN {X 0.070,Y -472.225,Z 777.493,A 0.000,B 0.000,C 90.000,E1 268.682} C_DIS
LIN {X -0.203,Y -466.380,Z 777.490,A 0.000,B 0.000,C 90.000,E1 268.224} C_DIS
LIN {X 0.055,Y -459.909,Z 777.488,A 0.000,B 0.000,C 90.000,E1 267.764} C_DIS
LIN {X 0.002,Y -456.678,Z 777.487,A 0.000,B 0.000,C 90.000,E1 267.593} C_DIS
LIN {X -0.051,Y -452.936,Z 777.486,A 0.000,B 0.000,C 90.000,E1 267.421} C_DIS
LIN {X -0.044,Y -445.410,Z 777.484,A 0.000,B 0.000,C 90.000,E1 267.135} C_DIS
LIN {X 0.027,Y -437.499,Z 777.483,A 0.000,B 0.000,C 90.000,E1 266.906} C_DIS
LIN {X 0.163,Y -428.001,Z 777.482,A 0.000,B 0.000,C 90.000,E1 266.731} C_DIS
LIN {X 0.105,Y -418.816,Z 777.482,A 0.000,B 0.000,C 90.000,E1 266.674} C_DIS
LIN {X 0.025,Y -180.962,Z 777.482,A 0.000,B 0.000,C 90.000,E1 266.674} C_DIS
LIN {X 0.060,Y -180.854,Z 777.472,A 0.000,B 0.000,C 90.000,E1 264.951} C_DIS
LIN {X -0.065,Y -178.966,Z 777.444,A 0.000,B 0.000,C 90.000,E1 259.926} C_DIS
LIN {X -0.055,Y -177.918,Z 777.435,A 0.000,B 0.000,C 90.000,E1 258.229} C_DIS
LIN {X -0.040,Y -175.554,Z 777.411,A 0.000,B 0.000,C 90.000,E1 253.976} C_DIS
LIN {X -0.033,Y -172.285,Z 777.387,A 0.000,B 0.000,C 90.000,E1 249.699} C_DIS
LIN {X -0.055,Y -171.764,Z 777.382,A 0.000,B 0.000,C 90.000,E1 248.847} C_DIS
LIN {X 0.024,Y -167.365,Z 777.354,A 0.000,B 0.000,C 90.000,E1 243.640} C_DIS
LIN {X -0.043,Y -166.754,Z 777.349,A 0.000,B 0.000,C 90.000,E1 242.794} C_DIS
LIN {X 0.018,Y -162.734,Z 777.325,A 0.000,B 0.000,C 90.000,E1 238.408} C_DIS
LIN {X 0.079,Y -161.424,Z 777.315,A 0.000,B 0.000,C 90.000,E1 236.628} C_DIS
LIN {X -0.102,Y -157.417,Z 777.290,A 0.000,B 0.000,C 90.000,E1 232.271} C_DIS
LIN {X 0.052,Y -155.420,Z 777.275,A 0.000,B 0.000,C 90.000,E1 229.542} C_DIS
LIN {X -0.017,Y -151.746,Z 777.250,A 0.000,B 0.000,C 90.000,E1 225.081} C_DIS
LIN {X -0.006,Y -149.944,Z 777.235,A 0.000,B 0.000,C 90.000,E1 222.366} C_DIS
LIN {X 0.022,Y -146.790,Z 777.210,A 0.000,B 0.000,C 90.000,E1 217.810} C_DIS
LIN {X -0.078,Y -145.364,Z 777.195,A 0.000,B 0.000,C 90.000,E1 215.105} C_DIS
LIN {X 0.039,Y -142.430,Z 777.164,A 0.000,B 0.000,C 90.000,E1 209.539} C_DIS
LIN {X -0.037,Y -141.420,Z 777.149,A 0.000,B 0.000,C 90.000,E1 206.796} C_DIS
LIN {X -0.056,Y -139.362,Z 777.113,A 0.000,B 0.000,C 90.000,E1 200.301} C_DIS
LIN {X 0.063,Y -138.806,Z 777.097,A 0.000,B 0.000,C 90.000,E1 197.457} C_DIS
LIN {X -0.018,Y -138.350,Z 777.056,A 0.000,B 0.000,C 90.000,E1 190.018} C_DIS
LIN {X -0.043,Y -139.545,Z 777.004,A 0.000,B 0.000,C 90.000,E1 180.688} C_DIS
LIN {X 0.050,Y -141.246,Z 776.973,A 0.000,B 0.000,C 90.000,E1 175.065} C_DIS
LIN {X 0.008,Y -142.616,Z 776.957,A 0.000,B 0.000,C 90.000,E1 172.299} C_DIS
LIN {X -0.039,Y -144.931,Z 776.932,A 0.000,B 0.000,C 90.000,E1 167.701} C_DIS
LIN {X -0.047,Y -147.560,Z 776.911,A 0.000,B 0.000,C 90.000,E1 164.031} C_DIS
LIN {X -0.016,Y -150.166,Z 776.891,A 0.000,B 0.000,C 90.000,E1 160.369} C_DIS
LIN {X -0.007,Y -153.541,Z 776.871,A 0.000,B 0.000,C 90.000,E1 156.741} C_DIS
LIN {X 0.045,Y -156.959,Z 776.851,A 0.000,B 0.000,C 90.000,E1 153.127} C_DIS
LIN {X -0.019,Y -161.066,Z 776.831,A 0.000,B 0.000,C 90.000,E1 149.587} C_DIS
LIN {X 0.066,Y -163.173,Z 776.821,A 0.000,B 0.000,C 90.000,E1 147.788} C_DIS
LIN {X 0.072,Y -167.593,Z 776.802,A 0.000,B 0.000,C 90.000,E1 144.276} C_DIS
LIN {X -0.018,Y -171.422,Z 776.787,A 0.000,B 0.000,C 90.000,E1 141.698} C_DIS
LIN {X 0.020,Y -176.340,Z 776.768,A 0.000,B 0.000,C 90.000,E1 138.243} C_DIS
LIN {X -0.112,Y -180.630,Z 776.754,A 0.000,B 0.000,C 90.000,E1 135.729} C_DIS
LIN {X 0.002,Y -186.031,Z 776.735,A 0.000,B 0.000,C 90.000,E1 132.324} C_DIS
LIN {X 0.065,Y -190.667,Z 776.721,A 0.000,B 0.000,C 90.000,E1 129.806} C_DIS
LIN {X 0.069,Y -192.422,Z 776.715,A 0.000,B 0.000,C 90.000,E1 128.749} C_DIS
LIN {X 0.070,Y -292.033,Z 776.715,A 0.000,B 0.000,C 90.000,E1 128.749} C_DIS
LIN {X -0.127,Y -294.207,Z 776.715,A 0.000,B 0.000,C 90.000,E1 128.749} C_DIS
LIN {X -0.074,Y -299.291,Z 776.714,A 0.000,B 0.000,C 90.000,E1 128.463} C_DIS
LIN {X -0.017,Y -302.054,Z 776.712,A 0.000,B 0.000,C 90.000,E1 128.177} C_DIS
LIN {X 0.022,Y -305.748,Z 776.709,A 0.000,B 0.000,C 90.000,E1 127.604} C_DIS
LIN {X -0.023,Y -307.248,Z 776.707,A 0.000,B 0.000,C 90.000,E1 127.282} C_DIS
LIN {X -0.009,Y -308.428,Z 776.705,A 0.000,B 0.000,C 90.000,E1 126.950} C_DIS
LIN {X 0.052,Y -319.383,Z 776.685,A 0.000,B 0.000,C 90.000,E1 123.372} C_DIS
LIN {X -0.133,Y -329.705,Z 776.670,A 0.000,B 0.000,C 90.000,E1 120.541} C_DIS
LIN {X -0.067,Y -341.370,Z 776.654,A 0.000,B 0.000,C 90.000,E1 117.719} C_DIS
LIN {X 0.007,Y -354.489,Z 776.639,A 0.000,B 0.000,C 90.000,E1 114.951} C_DIS
LIN {X -0.078,Y -367.460,Z 776.625,A 0.000,B 0.000,C 90.000,E1 112.567} C_DIS
LIN {X 0.098,Y -381.761,Z 776.612,A 0.000,B 0.000,C 90.000,E1 110.194} C_DIS
LIN {X -0.085,Y -397.497,Z 776.600,A 0.000,B 0.000,C 90.000,E1 107.928} C_DIS
LIN {X 0.124,Y -414.779,Z 776.587,A 0.000,B 0.000,C 90.000,E1 105.662} C_DIS
LIN {X 0.164,Y -433.734,Z 776.575,A 0.000,B 0.000,C 90.000,E1 103.480} C_DIS
LIN {X -0.208,Y -453.803,Z 776.564,A 0.000,B 0.000,C 90.000,E1 101.478} C_DIS
LIN {X 0.050,Y -466.616,Z 776.557,A 0.000,B 0.000,C 90.000,E1 100.254} C_DIS
LIN {X 0.077,Y -468.982,Z 776.556,A 0.000,B 0.000,C 90.000,E1 100.018} C_DIS
LIN {X -0.082,Y -470.853,Z 776.554,A 0.000,B 0.000,C 90.000,E1 99.792} C_DIS
LIN {X -0.161,Y -472.268,Z 776.553,A 0.000,B 0.000,C 90.000,E1 99.557} C_DIS
LIN {X 0.017,Y -474.152,Z 776.550,A 0.000,B 0.000,C 90.000,E1 99.029} C_DIS
LIN {X 0.129,Y -474.930,Z 776.547,A 0.000,B 0.000,C 90.000,E1 98.511} C_DIS
LIN {X -0.216,Y -474.737,Z 776.545,A 0.000,B 0.000,C 90.000,E1 98.049} C_DIS
LIN {X -0.084,Y -473.548,Z 776.542,A 0.000,B 0.000,C 90.000,E1 97.530} C_DIS
LIN {X -0.223,Y -472.524,Z 776.540,A 0.000,B 0.000,C 90.000,E1 97.296} C_DIS
LIN {X 0.105,Y -471.149,Z 776.539,A 0.000,B 0.000,C 90.000,E1 97.004} C_DIS
LIN {X 0.005,Y -451.841,Z 776.522,A 0.000,B 0.000,C 90.000,E1 93.955} C_DIS
LIN {X 0.083,Y -441.333,Z 776.512,A 0.000,B 0.000,C 90.000,E1 92.121} C_DIS
LIN {X -0.198,Y -432.144,Z 776.503,A 0.000,B 0.000,C 90.000,E1 90.573} C_DIS
LIN {X -0.212,Y -422.669,Z 776.494,A 0.000,B 0.000,C 90.000,E1 88.969} C_DIS
LIN {X 0.123,Y -411.452,Z 776.484,A 0.000,B 0.000,C 90.000,E1 87.020} C_DIS
LIN {X 0.178,Y -401.703,Z 776.474,A 0.000,B 0.000,C 90.000,E1 85.355} C_DIS
LIN {X 0.160,Y -388.718,Z 776.462,A 0.000,B 0.000,C 90.000,E1 83.109} C_DIS
LIN {X -0.043,Y -374.596,Z 776.448,A 0.000,B 0.000,C 90.000,E1 80.557} C_DIS
LIN {X 0.147,Y -356.573,Z 776.428,A 0.000,B 0.000,C 90.000,E1 76.992} C_DIS
LIN {X -0.171,Y -346.512,Z 776.416,A 0.000,B 0.000,C 90.000,E1 74.936} C_DIS
LIN {X 0.098,Y -333.719,Z 776.401,A 0.000,B 0.000,C 90.000,E1 72.127} C_DIS
LIN {X -0.048,Y -322.656,Z 776.387,A 0.000,B 0.000,C 90.000,E1 69.645} C_DIS
LIN {X 0.013,Y -309.456,Z 776.369,A 0.000,B 0.000,C 90.000,E1 66.433} C_DIS
LIN {X 0.048,Y -296.133,Z 776.349,A 0.000,B 0.000,C 90.000,E1 62.820} C_DIS
LIN {X 0.098,Y -285.125,Z 776.330,A 0.000,B 0.000,C 90.000,E1 59.459} C_DIS
LIN {X -0.009,Y -276.887,Z 776.315,A 0.000,B 0.000,C 90.000,E1 56.755} C_DIS
LIN {X -0.018,Y -268.849,Z 776.300,A 0.000,B 0.000,C 90.000,E1 53.989} C_DIS
LIN {X 0.025,Y -260.861,Z 776.284,A 0.000,B 0.000,C 90.000,E1 51.170} C_DIS
LIN {X -0.007,Y -252.992,Z 776.268,A 0.000,B 0.000,C 90.000,E1 48.324} C_DIS
LIN {X 0.070,Y -243.420,Z 776.248,A 0.000,B 0.000,C 90.000,E1 44.676} C_DIS
LIN {X -0.076,Y -235.947,Z 776.232,A 0.000,B 0.000,C 90.000,E1 41.757} C_DIS
LIN {X 0.050,Y -226.934,Z 776.211,A 0.000,B 0.000,C 90.000,E1 37.971} C_DIS
LIN {X 0.026,Y -218.454,Z 776.190,A 0.000,B 0.000,C 90.000,E1 34.151} C_DIS
LIN {X 0.033,Y -210.770,Z 776.168,A 0.000,B 0.000,C 90.000,E1 30.256} C_DIS
LIN {X -0.083,Y -205.353,Z 776.151,A 0.000,B 0.000,C 90.000,E1 27.129} C_DIS
LIN {X 0.093,Y -199.682,Z 776.128,A 0.000,B 0.000,C 90.000,E1 23.078} C_DIS
LIN {X 0.077,Y -195.123,Z 776.106,A 0.000,B 0.000,C 90.000,E1 19.033} C_DIS
LIN {X 0.046,Y -191.571,Z 776.083,A 0.000,B 0.000,C 90.000,E1 14.954} C_DIS
LIN {X -0.043,Y -188.463,Z 776.051,A 0.000,B 0.000,C 90.000,E1 9.208} C_DIS
LIN {X -0.017,Y -188.380,Z 775.979,A 0.000,B 0.000,C 90.000,E1 356.216} C_DIS
LIN {X -0.079,Y -191.348,Z 775.947,A 0.000,B 0.000,C 90.000,E1 350.443} C_DIS
LIN {X 0.041,Y -194.592,Z 775.924,A 0.000,B 0.000,C 90.000,E1 346.297} C_DIS
LIN {X -0.018,Y -198.837,Z 775.901,A 0.000,B 0.000,C 90.000,E1 342.236} C_DIS
LIN {X -0.062,Y -204.158,Z 775.879,A 0.000,B 0.000,C 90.000,E1 338.209} C_DIS
LIN {X -0.009,Y -210.390,Z 775.857,A 0.000,B 0.000,C 90.000,E1 334.204} C_DIS
LIN {X 0.042,Y -217.504,Z 775.835,A 0.000,B 0.000,C 90.000,E1 330.255} C_DIS
LIN {X 0.069,Y -225.314,Z 775.813,A 0.000,B 0.000,C 90.000,E1 326.373} C_DIS
LIN {X 0.093,Y -233.779,Z 775.792,A 0.000,B 0.000,C 90.000,E1 322.557} C_DIS
LIN {X -0.067,Y -243.013,Z 775.771,A 0.000,B 0.000,C 90.000,E1 318.852} C_DIS
LIN {X 0.015,Y -253.093,Z 775.751,A 0.000,B 0.000,C 90.000,E1 315.162} C_DIS
LIN {X -0.102,Y -264.006,Z 775.731,A 0.000,B 0.000,C 90.000,E1 311.595} C_DIS
LIN {X 0.038,Y -276.013,Z 775.711,A 0.000,B 0.000,C 90.000,E1 308.051} C_DIS
LIN {X 0.069,Y -289.298,Z 775.692,A 0.000,B 0.000,C 90.000,E1 304.612} C_DIS
LIN {X 0.068,Y -299.477,Z 775.679,A 0.000,B 0.000,C 90.000,E1 302.260} C_DIS
LIN {X -0.047,Y -316.108,Z 775.661,A 0.000,B 0.000,C 90.000,E1 298.999} C_DIS
LIN {X 0.086,Y -332.441,Z 775.645,A 0.000,B 0.000,C 90.000,E1 296.104} C_DIS
LIN {X -0.050,Y -342.083,Z 775.636,A 0.000,B 0.000,C 90.000,E1 294.567} C_DIS
LIN {X -0.188,Y -360.679,Z 775.621,A 0.000,B 0.000,C 90.000,E1 291.844} C_DIS
LIN {X -0.027,Y -378.827,Z 775.608,A 0.000,B 0.000,C 90.000,E1 289.450} C_DIS
LIN {X 0.013,Y -398.283,Z 775.595,A 0.000,B 0.000,C 90.000,E1 287.166} C_DIS
LIN {X 0.051,Y -413.229,Z 775.586,A 0.000,B 0.000,C 90.000,E1 285.481} C_DIS
LIN {X 0.021,Y -425.345,Z 775.578,A 0.000,B 0.000,C 90.000,E1 284.120} C_DIS
LIN {X 0.030,Y -437.127,Z 775.571,A 0.000,B 0.000,C 90.000,E1 282.771} C_DIS
LIN {X -0.210,Y -448.465,Z 775.564,A 0.000,B 0.000,C 90.000,E1 281.478} C_DIS
LIN {X -0.117,Y -456.936,Z 775.558,A 0.000,B 0.000,C 90.000,E1 280.423} C_DIS
LIN {X -0.008,Y -464.854,Z 775.552,A 0.000,B 0.000,C 90.000,E1 279.378} C_DIS
LIN {X 0.130,Y -472.342,Z 775.546,A 0.000,B 0.000,C 90.000,E1 278.341} C_DIS
LIN {X -0.044,Y -479.067,Z 775.541,A 0.000,B 0.000,C 90.000,E1 277.352} C_DIS
LIN {X -0.087,Y -483.346,Z 775.537,A 0.000,B 0.000,C 90.000,E1 276.606} C_DIS
LIN {X -0.031,Y -486.863,Z 775.532,A 0.000,B 0.000,C 90.000,E1 275.853} C_DIS
LIN {X 0.003,Y -489.549,Z 775.528,A 0.000,B 0.000,C 90.000,E1 275.106} C_DIS
LIN {X 0.212,Y -490.916,Z 775.526,A 0.000,B 0.000,C 90.000,E1 274.588} C_DIS
LIN {X -0.096,Y -491.901,Z 775.523,A 0.000,B 0.000,C 90.000,E1 274.131} C_DIS
LIN {X 0.130,Y -492.498,Z 775.520,A 0.000,B 0.000,C 90.000,E1 273.612} C_DIS
LIN {X -0.134,Y -492.696,Z 775.517,A 0.000,B 0.000,C 90.000,E1 273.151} C_DIS
LIN {X 0.071,Y -492.438,Z 775.515,A 0.000,B 0.000,C 90.000,E1 272.636} C_DIS
LIN {X -0.212,Y -491.789,Z 775.512,A 0.000,B 0.000,C 90.000,E1 272.178} C_DIS
LIN {X 0.013,Y -490.697,Z 775.509,A 0.000,B 0.000,C 90.000,E1 271.661} C_DIS
LIN {X 0.215,Y -489.099,Z 775.507,A 0.000,B 0.000,C 90.000,E1 271.146} C_DIS
LIN {X -0.074,Y -487.055,Z 775.504,A 0.000,B 0.000,C 90.000,E1 270.688} C_DIS
LIN {X 0.115,Y -484.444,Z 775.501,A 0.000,B 0.000,C 90.000,E1 270.172} C_DIS
LIN {X -0.199,Y -481.212,Z 775.498,A 0.000,B 0.000,C 90.000,E1 269.714} C_DIS
LIN {X -0.046,Y -477.272,Z 775.495,A 0.000,B 0.000,C 90.000,E1 269.198} C_DIS
LIN {X 0.083,Y -472.421,Z 775.493,A 0.000,B 0.000,C 90.000,E1 268.682} C_DIS
LIN {X -0.154,Y -466.655,Z 775.490,A 0.000,B 0.000,C 90.000,E1 268.224} C_DIS
LIN {X -0.021,Y -463.649,Z 775.489,A 0.000,B 0.000,C 90.000,E1 267.993} C_DIS
LIN {X 0.030,Y -457.026,Z 775.487,A 0.000,B 0.000,C 90.000,E1 267.593} C_DIS
LIN {X 0.186,Y -449.841,Z 775.485,A 0.000,B 0.000,C 90.000,E1 267.249} C_DIS
LIN {X -0.031,Y -442.229,Z 775.483,A 0.000,B 0.000,C 90.000,E1 267.020} C_DIS
LIN {X -0.166,Y -433.742,Z 775.482,A 0.000,B 0.000,C 90.000,E1 266.846} C_DIS
LIN {X 0.186,Y -423.489,Z 775.482,A 0.000,B 0.000,C 90.000,E1 266.674} C_DIS
LIN {X -0.009,Y -418.245,Z 775.482,A 0.000,B 0.000,C 90.000,E1 266.674} C_DIS
LIN {X -0.025,Y -180.961,Z 775.482,A 0.000,B 0.000,C 90.000,E1 266.674} C_DIS
LIN {X 0.017,Y -180.886,Z 775.473,A 0.000,B 0.000,C 90.000,E1 265.122} C_DIS
LIN {X 0.043,Y -179.092,Z 775.447,A 0.000,B 0.000,C 90.000,E1 260.387} C_DIS
LIN {X -0.038,Y -178.823,Z 775.442,A 0.000,B 0.000,C 90.000,E1 259.567} C_DIS
LIN {X 0.043,Y -175.868,Z 775.414,A 0.000,B 0.000,C 90.000,E1 254.448} C_DIS
LIN {X 0.037,Y -173.838,Z 775.399,A 0.000,B 0.000,C 90.000,E1 251.891} C_DIS
LIN {X 0.027,Y -171.507,Z 775.380,A 0.000,B 0.000,C 90.000,E1 248.465} C_DIS
LIN {X 0.014,Y -167.734,Z 775.356,A 0.000,B 0.000,C 90.000,E1 244.152} C_DIS
LIN {X 0.029,Y -166.431,Z 775.347,A 0.000,B 0.000,C 90.000,E1 242.410} C_DIS
LIN {X -0.057,Y -163.150,Z 775.327,A 0.000,B 0.000,C 90.000,E1 238.948} C_DIS
LIN {X -0.007,Y -161.107,Z 775.313,A 0.000,B 0.000,C 90.000,E1 236.294} C_DIS
LIN {X -0.025,Y -157.833,Z 775.293,A 0.000,B 0.000,C 90.000,E1 232.763} C_DIS
LIN {X 0.039,Y -155.866,Z 775.278,A 0.000,B 0.000,C 90.000,E1 230.070} C_DIS
LIN {X -0.012,Y -152.116,Z 775.253,A 0.000,B 0.000,C 90.000,E1 225.607} C_DIS
LIN {X 0.002,Y -150.366,Z 775.238,A 0.000,B 0.000,C 90.000,E1 222.894} C_DIS
LIN {X -0.076,Y -147.101,Z 775.213,A 0.000,B 0.000,C 90.000,E1 218.382} C_DIS
LIN {X 0.035,Y -145.669,Z 775.198,A 0.000,B 0.000,C 90.000,E1 215.598} C_DIS
LIN {X 0.038,Y -143.052,Z 775.172,A 0.000,B 0.000,C 90.000,E1 211.003} C_DIS
LIN {X -0.027,Y -141.674,Z 775.152,A 0.000,B 0.000,C 90.000,E1 207.334} C_DIS
LIN {X -0.048,Y -139.454,Z 775.116,A 0.000,B 0.000,C 90.000,E1 200.844} C_DIS
LIN {X 0.003,Y -139.188,Z 775.105,A 0.000,B 0.000,C 90.000,E1 198.960} C_DIS
LIN {X 0.025,Y -138.323,Z 775.053,A 0.000,B 0.000,C 90.000,E1 189.613} C_DIS
LIN {X 0.033,Y -139.458,Z 775.007,A 0.000,B 0.000,C 90.000,E1 181.203} C_DIS
LIN {X -0.026,Y -141.012,Z 774.976,A 0.000,B 0.000,C 90.000,E1 175.641} C_DIS
LIN {X 0.064,Y -142.765,Z 774.955,A 0.000,B 0.000,C 90.000,E1 171.894} C_DIS
LIN {X 0.019,Y -145.174,Z 774.929,A 0.000,B 0.000,C 90.000,E1 167.297} C_DIS
LIN {X 0.053,Y -147.796,Z 774.909,A 0.000,B 0.000,C 90.000,E1 163.614} C_DIS
LIN {X -0.052,Y -150.479,Z 774.889,A 0.000,B 0.000,C 90.000,E1 160.007} C_DIS
LIN {X 0.022,Y -153.934,Z 774.869,A 0.000,B 0.000,C 90.000,E1 156.357} C_DIS
LIN {X 0.085,Y -157.344,Z 774.849,A 0.000,B 0.000,C 90.000,E1 152.743} C_DIS
LIN {X 0.029,Y -161.539,Z 774.829,A 0.000,B 0.000,C 90.000,E1 149.203} C_DIS
LIN {X 0.041,Y -165.736,Z 774.809,A 0.000,B 0.000,C 90.000,E1 145.674} C_DIS
LIN {X 0.029,Y -170.688,Z 774.790,A 0.000,B 0.000,C 90.000,E1 142.190} C_DIS
LIN {X -0.060,Y -175.563,Z 774.771,A 0.000,B 0.000,C 90.000,E1 138.771} C_DIS
LIN {X 0.061,Y -181.181,Z 774.752,A 0.000,B 0.000,C 90.000,E1 135.324} C_DIS
LIN {X -0.070,Y -186.639,Z 774.733,A 0.000,B 0.000,C 90.000,E1 132.000} C_DIS
LIN {X -0.064,Y -191.479,Z 774.719,A 0.000,B 0.000,C 90.000,E1 129.358} C_DIS
LIN {X 0.113,Y -192.400,Z 774.715,A 0.000,B 0.000,C 90.000,E1 128.749} C_DIS
LIN {X 0.137,Y -292.127,Z 774.715,A 0.000,B 0.000,C 90.000,E1 128.749} C_DIS
LIN {X -0.064,Y -296.272,Z 774.715,A 0.000,B 0.000,C 90.000,E1 128.669} C_DIS
LIN {X 0.045,Y -299.124,Z 774.714,A 0.000,B 0.000,C 90.000,E1 128.463} C_DIS
LIN {X -0.091,Y -302.852,Z 774.712,A 0.000,B 0.000,C 90.000,E1 128.096} C_DIS
LIN {X -0.182,Y -306.334,Z 774.708,A 0.000,B 0.000,C 90.000,E1 127.523} C_DIS
LIN {X 0.020,Y -307.695,Z 774.706,A 0.000,B 0.000,C 90.000,E1 127.156} C_DIS
LIN {X 0.040,Y -310.627,Z 774.701,A 0.000,B 0.000,C 90.000,E1 126.171} C_DIS
LIN {X -0.076,Y -320.839,Z 774.683,A 0.000,B 0.000,C 90.000,E1 122.959} C_DIS
LIN {X 0.063,Y -331.357,Z 774.667,A 0.000,B 0.000,C 90.000,E1 120.079} C_DIS
LIN {X 0.178,Y -343.237,Z 774.652,A 0.000,B 0.000,C 90.000,E1 117.257} C_DIS
LIN {X 0.164,Y -356.580,Z 774.636,A 0.000,B 0.000,C 90.000,E1 114.515} C_DIS
LIN {X -0.001,Y -369.771,Z 774.623,A 0.000,B 0.000,C 90.000,E1 112.153} C_DIS
LIN {X 0.020,Y -384.308,Z 774.610,A 0.000,B 0.000,C 90.000,E1 109.812} C_DIS
LIN {X 0.141,Y -400.297,Z 774.597,A 0.000,B 0.000,C 90.000,E1 107.511} C_DIS
LIN {X 0.032,Y -417.854,Z 774.585,A 0.000,B 0.000,C 90.000,E1 105.300} C_DIS
LIN {X 0.166,Y -437.072,Z 774.573,A 0.000,B 0.000,C 90.000,E1 103.119} C_DIS
LIN {X -0.070,Y -457.240,Z 774.562,A 0.000,B 0.000,C 90.000,E1 101.130} C_DIS
LIN {X -0.181,Y -467.524,Z 774.557,A 0.000,B 0.000,C 90.000,E1 100.197} C_DIS
LIN {X -0.147,Y -469.665,Z 774.555,A 0.000,B 0.000,C 90.000,E1 99.962} C_DIS
LIN {X 0.164,Y -471.426,Z 774.554,A 0.000,B 0.000,C 90.000,E1 99.670} C_DIS
LIN {X -0.066,Y -472.748,Z 774.552,A 0.000,B 0.000,C 90.000,E1 99.443} C_DIS
LIN {X 0.117,Y -474.399,Z 774.550,A 0.000,B 0.000,C 90.000,E1 98.916} C_DIS
LIN {X -0.237,Y -474.987,Z 774.547,A 0.000,B 0.000,C 90.000,E1 98.454} C_DIS
LIN {X -0.109,Y -474.610,Z 774.544,A 0.000,B 0.000,C 90.000,E1 97.936} C_DIS
LIN {X 0.085,Y -473.215,Z 774.541,A 0.000,B 0.000,C 90.000,E1 97.409} C_DIS
LIN {X -0.115,Y -472.065,Z 774.540,A 0.000,B 0.000,C 90.000,E1 97.182} C_DIS
LIN {X 0.113,Y -465.562,Z 774.534,A 0.000,B 0.000,C 90.000,E1 96.144} C_DIS
LIN {X -0.148,Y -449.765,Z 774.520,A 0.000,B 0.000,C 90.000,E1 93.612} C_DIS
LIN {X -0.085,Y -439.279,Z 774.510,A 0.000,B 0.000,C 90.000,E1 91.776} C_DIS
LIN {X 0.020,Y -429.991,Z 774.501,A 0.000,B 0.000,C 90.000,E1 90.172} C_DIS
LIN {X -0.036,Y -420.477,Z 774.492,A 0.000,B 0.000,C 90.000,E1 88.568} C_DIS
LIN {X 0.161,Y -410.876,Z 774.483,A 0.000,B 0.000,C 90.000,E1 86.906} C_DIS
LIN {X -0.117,Y -399.471,Z 774.472,A 0.000,B 0.000,C 90.000,E1 85.008} C_DIS
LIN {X -0.171,Y -386.575,Z 774.460,A 0.000,B 0.000,C 90.000,E1 82.761} C_DIS
LIN {X -0.042,Y -372.490,Z 774.445,A 0.000,B 0.000,C 90.000,E1 80.151} C_DIS
LIN {X 0.109,Y -356.086,Z 774.427,A 0.000,B 0.000,C 90.000,E1 76.881} C_DIS
LIN {X -0.133,Y -346.023,Z 774.415,A 0.000,B 0.000,C 90.000,E1 74.810} C_DIS
LIN {X -0.174,Y -334.685,Z 774.402,A 0.000,B 0.000,C 90.000,E1 72.362} C_DIS
LIN {X -0.026,Y -322.261,Z 774.386,A 0.000,B 0.000,C 90.000,E1 69.518} C_DIS
LIN {X 0.067,Y -307.876,Z 774.367,A 0.000,B 0.000,C 90.000,E1 65.973} C_DIS
LIN {X 0.055,Y -294.762,Z 774.346,A 0.000,B 0.000,C 90.000,E1 62.359} C_DIS
LIN {X 0.094,Y -284.970,Z 774.330,A 0.000,B 0.000,C 90.000,E1 59.331} C_DIS
LIN {X -0.019,Y -276.803,Z 774.315,A 0.000,B 0.000,C 90.000,E1 56.628} C_DIS
LIN {X -0.034,Y -268.805,Z 774.299,A 0.000,B 0.000,C 90.000,E1 53.863} C_DIS
LIN {X 0.042,Y -262.857,Z 774.288,A 0.000,B 0.000,C 90.000,E1 51.743} C_DIS
LIN {X -0.102,Y -254.969,Z 774.272,A 0.000,B 0.000,C 90.000,E1 48.933} C_DIS
LIN {X -0.132,Y -247.234,Z 774.256,A 0.000,B 0.000,C 90.000,E1 46.053} C_DIS
LIN {X -0.013,Y -239.735,Z 774.239,A 0.000,B 0.000,C 90.000,E1 43.095} C_DIS
LIN {X 0.100,Y -232.312,Z 774.223,A 0.000,B 0.000,C 90.000,E1 40.092} C_DIS
LIN {X 0.075,Y -225.221,Z 774.206,A 0.000,B 0.000,C 90.000,E1 37.076} C_DIS
LIN {X 0.044,Y -216.875,Z 774.185,A 0.000,B 0.000,C 90.000,E1 33.245} C_DIS
LIN {X 0.031,Y -210.825,Z 774.167,A 0.000,B 0.000,C 90.000,E1 30.129} C_DIS
LIN {X -0.082,Y -205.427,Z 774.150,A 0.000,B 0.000,C 90.000,E1 27.001} C_DIS
LIN {X 0.095,Y -199.763,Z 774.128,A 0.000,B 0.000,C 90.000,E1 22.950} C_DIS
LIN {X 0.080,Y -195.218,Z 774.105,A 0.000,B 0.000,C 90.000,E1 18.906} C_DIS
LIN {X 0.047,Y -191.690,Z 774.082,A 0.000,B 0.000,C 90.000,E1 14.828} C_DIS
LIN {X -0.078,Y -188.593,Z 774.050,A 0.000,B 0.000,C 90.000,E1 9.095} C_DIS
LIN {X -0.014,Y -188.509,Z 773.979,A 0.000,B 0.000,C 90.000,E1 356.216} C_DIS
LIN {X -0.071,Y -191.472,Z 773.947,A 0.000,B 0.000,C 90.000,E1 350.443} C_DIS
LIN {X 0.055,Y -194.706,Z 773.924,A 0.000,B 0.000,C 90.000,E1 346.297} C_DIS
LIN {X -0.001,Y -198.981,Z 773.901,A 0.000,B 0.000,C 90.000,E1 342.236} C_DIS
LIN {X -0.040,Y -204.299,Z 773.879,A 0.000,B 0.000,C 90.000,E1 338.209} C_DIS
LIN {X 0.018,Y -210.520,Z 773.857,A 0.000,B 0.000,C 90.000,E1 334.204} C_DIS
LIN {X 0.073,Y -217.622,Z 773.835,A 0.000,B 0.000,C 90.000,E1 330.255} C_DIS
LIN {X -0.081,Y -225.429,Z 773.813,A 0.000,B 0.000,C 90.000,E1 326.421} C_DIS
LIN {X 0.135,Y -233.867,Z 773.792,A 0.000,B 0.000,C 90.000,E1 322.557} C_DIS
LIN {X -0.021,Y -243.071,Z 773.771,A 0.000,B 0.000,C 90.000,E1 318.852} C_DIS
LIN {X -0.119,Y -252.089,Z 773.753,A 0.000,B 0.000,C 90.000,E1 315.567} C_DIS
LIN {X 0.101,Y -262.894,Z 773.733,A 0.000,B 0.000,C 90.000,E1 311.919} C_DIS
LIN {X 0.003,Y -274.783,Z 773.713,A 0.000,B 0.000,C 90.000,E1 308.418} C_DIS
LIN {X -0.004,Y -287.911,Z 773.694,A 0.000,B 0.000,C 90.000,E1 304.978} C_DIS
LIN {X -0.036,Y -297.898,Z 773.681,A 0.000,B 0.000,C 90.000,E1 302.625} C_DIS
LIN {X -0.203,Y -307.532,Z 773.670,A 0.000,B 0.000,C 90.000,E1 300.669} C_DIS
LIN {X 0.063,Y -324.980,Z 773.652,A 0.000,B 0.000,C 90.000,E1 297.385} C_DIS
LIN {X -0.117,Y -339.981,Z 773.638,A 0.000,B 0.000,C 90.000,E1 294.899} C_DIS
LIN {X 0.086,Y -354.235,Z 773.626,A 0.000,B 0.000,C 90.000,E1 292.717} C_DIS
LIN {X 0.069,Y -367.168,Z 773.616,A 0.000,B 0.000,C 90.000,E1 290.918} C_DIS
LIN {X -0.077,Y -388.280,Z 773.602,A 0.000,B 0.000,C 90.000,E1 288.308} C_DIS
LIN {X -0.052,Y -403.024,Z 773.592,A 0.000,B 0.000,C 90.000,E1 286.622} C_DIS
LIN {X -0.159,Y -415.406,Z 773.585,A 0.000,B 0.000,C 90.000,E1 285.245} C_DIS
LIN {X -0.170,Y -427.463,Z 773.577,A 0.000,B 0.000,C 90.000,E1 283.883} C_DIS
LIN {X -0.128,Y -439.091,Z 773.570,A 0.000,B 0.000,C 90.000,E1 282.535} C_DIS
LIN {X -0.141,Y -448.135,Z 773.564,A 0.000,B 0.000,C 90.000,E1 281.478} C_DIS
LIN {X -0.051,Y -456.622,Z 773.558,A 0.000,B 0.000,C 90.000,E1 280.423} C_DIS
LIN {X 0.055,Y -464.551,Z 773.552,A 0.000,B 0.000,C 90.000,E1 279.378} C_DIS
LIN {X 0.191,Y -472.070,Z 773.546,A 0.000,B 0.000,C 90.000,E1 278.341} C_DIS
LIN {X 0.152,Y -477.245,Z 773.542,A 0.000,B 0.000,C 90.000,E1 277.587} C_DIS
LIN {X 0.160,Y -481.813,Z 773.538,A 0.000,B 0.000,C 90.000,E1 276.834} C_DIS
LIN {X 0.148,Y -485.665,Z 773.534,A 0.000,B 0.000,C 90.000,E1 276.087} C_DIS
LIN {X -0.145,Y -487.764,Z 773.531,A 0.000,B 0.000,C 90.000,E1 275.625} C_DIS
LIN {X 0.058,Y -489.500,Z 773.528,A 0.000,B 0.000,C 90.000,E1 275.106} C_DIS
LIN {X -0.221,Y -490.900,Z 773.526,A 0.000,B 0.000,C 90.000,E1 274.645} C_DIS
LIN {X -0.040,Y -491.928,Z 773.523,A 0.000,B 0.000,C 90.000,E1 274.131} C_DIS
LIN {X 0.186,Y -492.546,Z 773.520,A 0.000,B 0.000,C 90.000,E1 273.612} C_DIS
LIN {X -0.105,Y -492.786,Z 773.517,A 0.000,B 0.000,C 90.000,E1 273.154} C_DIS
LIN {X 0.127,Y -492.539,Z 773.515,A 0.000,B 0.000,C 90.000,E1 272.636} C_DIS
LIN {X -0.155,Y -491.920,Z 773.512,A 0.000,B 0.000,C 90.000,E1 272.178} C_DIS
LIN {X 0.070,Y -490.844,Z 773.509,A 0.000,B 0.000,C 90.000,E1 271.661} C_DIS
LIN {X -0.216,Y -489.312,Z 773.507,A 0.000,B 0.000,C 90.000,E1 271.203} C_DIS
LIN {X -0.017,Y -487.281,Z 773.504,A 0.000,B 0.000,C 90.000,E1 270.688} C_DIS
LIN {X 0.173,Y -484.700,Z 773.501,A 0.000,B 0.000,C 90.000,E1 270.172} C_DIS
LIN {X -0.139,Y -481.490,Z 773.498,A 0.000,B 0.000,C 90.000,E1 269.714} C_DIS
LIN {X 0.015,Y -477.526,Z 773.496,A 0.000,B 0.000,C 90.000,E1 269.198} C_DIS
LIN {X 0.145,Y -472.716,Z 773.493,A 0.000,B 0.000,C 90.000,E1 268.682} C_DIS
LIN {X -0.142,Y -466.877,Z 773.490,A 0.000,B 0.000,C 90.000,E1 268.224} C_DIS
LIN {X 0.099,Y -460.518,Z 773.488,A 0.000,B 0.000,C 90.000,E1 267.764} C_DIS
LIN {X -0.061,Y -453.556,Z 773.486,A 0.000,B 0.000,C 90.000,E1 267.421} C_DIS
LIN {X -0.102,Y -446.137,Z 773.484,A 0.000,B 0.000,C 90.000,E1 267.135} C_DIS
LIN {X -0.084,Y -438.049,Z 773.483,A 0.000,B 0.000,C 90.000,E1 266.906} C_DIS
LIN {X 0.028,Y -428.557,Z 773.482,A 0.000,B 0.000,C 90.000,E1 266.731} C_DIS
LIN {X -0.080,Y -419.112,Z 773.481,A 0.000,B 0.000,C 90.000,E1 266.674} C_DIS
LIN {X -0.056,Y -180.960,Z 773.481,A 0.000,B 0.000,C 90.000,E1 266.674} C_DIS
LIN {X -0.015,Y -180.884,Z 773.473,A 0.000,B 0.000,C 90.000,E1 265.122} C_DIS
LIN {X -0.071,Y -178.818,Z 773.442,A 0.000,B 0.000,C 90.000,E1 259.567} C_DIS
LIN {X 0.012,Y -175.863,Z 773.414,A 0.000,B 0.000,C 90.000,E1 254.448} C_DIS
LIN {X 0.060,Y -173.830,Z 773.399,A 0.000,B 0.000,C 90.000,E1 251.873} C_DIS
LIN {X -0.005,Y -171.498,Z 773.380,A 0.000,B 0.000,C 90.000,E1 248.465} C_DIS
LIN {X -0.018,Y -167.726,Z 773.356,A 0.000,B 0.000,C 90.000,E1 244.152} C_DIS
LIN {X -0.001,Y -166.421,Z 773.347,A 0.000,B 0.000,C 90.000,E1 242.410} C_DIS
LIN {X -0.003,Y -163.141,Z 773.327,A 0.000,B 0.000,C 90.000,E1 238.918} C_DIS
LIN {X -0.038,Y -161.097,Z 773.313,A 0.000,B 0.000,C 90.000,E1 236.294} C_DIS
LIN {X -0.054,Y -157.824,Z 773.293,A 0.000,B 0.000,C 90.000,E1 232.763} C_DIS
LIN {X 0.010,Y -155.859,Z 773.278,A 0.000,B 0.000,C 90.000,E1 230.070} C_DIS
LIN {X 0.065,Y -152.108,Z 773.253,A 0.000,B 0.000,C 90.000,E1 225.567} C_DIS
LIN {X -0.027,Y -150.358,Z 773.238,A 0.000,B 0.000,C 90.000,E1 222.894} C_DIS
LIN {X 0.012,Y -147.094,Z 773.213,A 0.000,B 0.000,C 90.000,E1 218.338} C_DIS
LIN {X 0.006,Y -145.665,Z 773.198,A 0.000,B 0.000,C 90.000,E1 215.598} C_DIS
LIN {X 0.010,Y -143.047,Z 773.172,A 0.000,B 0.000,C 90.000,E1 211.003} C_DIS
LIN {X 0.010,Y -141.670,Z 773.152,A 0.000,B 0.000,C 90.000,E1 207.308} C_DIS
LIN {X 0.055,Y -139.452,Z 773.116,A 0.000,B 0.000,C 90.000,E1 200.791} C_DIS
LIN {X -0.024,Y -139.186,Z 773.105,A 0.000,B 0.000,C 90.000,E1 198.960} C_DIS
LIN {X -0.002,Y -138.322,Z 773.053,A 0.000,B 0.000,C 90.000,E1 189.613} C_DIS
LIN {X 0.006,Y -139.460,Z 773.007,A 0.000,B 0.000,C 90.000,E1 181.203} C_DIS
LIN {X -0.054,Y -141.016,Z 772.976,A 0.000,B 0.000,C 90.000,E1 175.641} C_DIS
LIN {X 0.036,Y -142.770,Z 772.955,A 0.000,B 0.000,C 90.000,E1 171.894} C_DIS
LIN {X -0.009,Y -145.180,Z 772.929,A 0.000,B 0.000,C 90.000,E1 167.297} C_DIS
LIN {X 0.025,Y -147.803,Z 772.909,A 0.000,B 0.000,C 90.000,E1 163.614} C_DIS
LIN {X -0.080,Y -150.489,Z 772.889,A 0.000,B 0.000,C 90.000,E1 160.007} C_DIS
LIN {X -0.008,Y -153.944,Z 772.869,A 0.000,B 0.000,C 90.000,E1 156.357} C_DIS
LIN {X 0.055,Y -157.356,Z 772.849,A 0.000,B 0.000,C 90.000,E1 152.743} C_DIS
LIN {X -0.001,Y -161.552,Z 772.829,A 0.000,B 0.000,C 90.000,E1 149.203} C_DIS
LIN {X 0.010,Y -165.750,Z 772.809,A 0.000,B 0.000,C 90.000,E1 145.674} C_DIS
LIN {X -0.003,Y -170.705,Z 772.790,A 0.000,B 0.000,C 90.000,E1 142.190} C_DIS
LIN {X -0.091,Y -175.578,Z 772.771,A 0.000,B 0.000,C 90.000,E1 138.771} C_DIS
LIN {X 0.028,Y -181.196,Z 772.752,A 0.000,B 0.000,C 90.000,E1 135.324} C_DIS
LIN {X 0.022,Y -186.658,Z 772.733,A 0.000,B 0.000,C 90.000,E1 131.962} C_DIS
LIN {X 0.025,Y -191.495,Z 772.719,A 0.000,B 0.000,C 90.000,E1 129.322} C_DIS
LIN {X -0.094,Y -192.367,Z 772.716,A 0.000,B 0.000,C 90.000,E1 128.830} C_DIS
LIN {X -0.176,Y -291.552,Z 772.716,A 0.000,B 0.000,C 90.000,E1 128.830} C_DIS
LIN {X -0.116,Y -296.702,Z 772.715,A 0.000,B 0.000,C 90.000,E1 128.669} C_DIS
LIN {X -0.006,Y -299.370,Z 772.714,A 0.000,B 0.000,C 90.000,E1 128.463} C_DIS
LIN {X 0.156,Y -303.152,Z 772.711,A 0.000,B 0.000,C 90.000,E1 128.016} C_DIS
LIN {X 0.058,Y -305.074,Z 772.710,A 0.000,B 0.000,C 90.000,E1 127.729} C_DIS
LIN {X -0.041,Y -306.586,Z 772.708,A 0.000,B 0.000,C 90.000,E1 127.443} C_DIS
LIN {X 0.166,Y -307.875,Z 772.706,A 0.000,B 0.000,C 90.000,E1 127.076} C_DIS
LIN {X 0.011,Y -319.900,Z 772.685,A 0.000,B 0.000,C 90.000,E1 123.214} C_DIS
LIN {X 0.114,Y -330.296,Z 772.669,A 0.000,B 0.000,C 90.000,E1 120.335} C_DIS
LIN {X 0.201,Y -342.042,Z 772.653,A 0.000,B 0.000,C 90.000,E1 117.513} C_DIS
LIN {X 0.149,Y -355.246,Z 772.638,A 0.000,B 0.000,C 90.000,E1 114.771} C_DIS
LIN {X 0.093,Y -368.301,Z 772.624,A 0.000,B 0.000,C 90.000,E1 112.386} C_DIS
LIN {X -0.059,Y -382.692,Z 772.611,A 0.000,B 0.000,C 90.000,E1 110.066} C_DIS
LIN {X 0.027,Y -398.523,Z 772.599,A 0.000,B 0.000,C 90.000,E1 107.764} C_DIS
LIN {X -0.118,Y -415.909,Z 772.586,A 0.000,B 0.000,C 90.000,E1 105.552} C_DIS
LIN {X 0.047,Y -434.978,Z 772.574,A 0.000,B 0.000,C 90.000,E1 103.355} C_DIS
LIN {X 0.197,Y -455.086,Z 772.563,A 0.000,B 0.000,C 90.000,E1 101.299} C_DIS
LIN {X -0.027,Y -467.891,Z 772.556,A 0.000,B 0.000,C 90.000,E1 100.141} C_DIS
LIN {X 0.011,Y -469.943,Z 772.555,A 0.000,B 0.000,C 90.000,E1 99.905} C_DIS
LIN {X -0.140,Y -471.639,Z 772.554,A 0.000,B 0.000,C 90.000,E1 99.670} C_DIS
LIN {X 0.173,Y -472.912,Z 772.552,A 0.000,B 0.000,C 90.000,E1 99.378} C_DIS
LIN {X -0.188,Y -474.488,Z 772.549,A 0.000,B 0.000,C 90.000,E1 98.916} C_DIS
LIN {X -0.070,Y -475.014,Z 772.547,A 0.000,B 0.000,C 90.000,E1 98.398} C_DIS
LIN {X 0.124,Y -474.575,Z 772.544,A 0.000,B 0.000,C 90.000,E1 97.871} C_DIS
LIN {X -0.216,Y -473.108,Z 772.541,A 0.000,B 0.000,C 90.000,E1 97.409} C_DIS
LIN {X 0.053,Y -471.915,Z 772.540,A 0.000,B 0.000,C 90.000,E1 97.125} C_DIS
LIN {X -0.034,Y -458.860,Z 772.528,A 0.000,B 0.000,C 90.000,E1 95.106} C_DIS
LIN {X 0.126,Y -442.093,Z 772.513,A 0.000,B 0.000,C 90.000,E1 92.236} C_DIS
LIN {X -0.143,Y -432.951,Z 772.504,A 0.000,B 0.000,C 90.000,E1 90.688} C_DIS
LIN {X -0.143,Y -423.491,Z 772.495,A 0.000,B 0.000,C 90.000,E1 89.083} C_DIS
LIN {X -0.208,Y -412.301,Z 772.484,A 0.000,B 0.000,C 90.000,E1 87.192} C_DIS
LIN {X -0.128,Y -402.565,Z 772.475,A 0.000,B 0.000,C 90.000,E1 85.527} C_DIS
LIN {X -0.110,Y -389.620,Z 772.463,A 0.000,B 0.000,C 90.000,E1 83.280} C_DIS
LIN {X 0.049,Y -373.891,Z 772.447,A 0.000,B 0.000,C 90.000,E1 80.387} C_DIS
LIN {X -0.105,Y -357.395,Z 772.429,A 0.000,B 0.000,C 90.000,E1 77.173} C_DIS
LIN {X 0.019,Y -347.372,Z 772.417,A 0.000,B 0.000,C 90.000,E1 75.046} C_DIS
LIN {X 0.008,Y -336.007,Z 772.403,A 0.000,B 0.000,C 90.000,E1 72.598} C_DIS
LIN {X 0.194,Y -323.566,Z 772.388,A 0.000,B 0.000,C 90.000,E1 69.752} C_DIS
LIN {X -0.080,Y -309.128,Z 772.368,A 0.000,B 0.000,C 90.000,E1 66.282} C_DIS
LIN {X -0.034,Y -295.963,Z 772.348,A 0.000,B 0.000,C 90.000,E1 62.666} C_DIS
LIN {X -0.072,Y -287.231,Z 772.333,A 0.000,B 0.000,C 90.000,E1 59.999} C_DIS
LIN {X 0.024,Y -276.999,Z 772.314,A 0.000,B 0.000,C 90.000,E1 56.580} C_DIS
LIN {X -0.053,Y -269.055,Z 772.299,A 0.000,B 0.000,C 90.000,E1 53.829} C_DIS
LIN {X 0.000,Y -261.145,Z 772.283,A 0.000,B 0.000,C 90.000,E1 51.009} C_DIS
LIN {X -0.022,Y -253.343,Z 772.268,A 0.000,B 0.000,C 90.000,E1 48.162} C_DIS
LIN {X 0.069,Y -243.792,Z 772.247,A 0.000,B 0.000,C 90.000,E1 44.514} C_DIS
LIN {X -0.013,Y -238.151,Z 772.235,A 0.000,B 0.000,C 90.000,E1 42.324} C_DIS
LIN {X -0.091,Y -230.778,Z 772.219,A 0.000,B 0.000,C 90.000,E1 39.358} C_DIS
LIN {X 0.032,Y -223.770,Z 772.202,A 0.000,B 0.000,C 90.000,E1 36.297} C_DIS
LIN {X -0.046,Y -215.539,Z 772.180,A 0.000,B 0.000,C 90.000,E1 32.467} C_DIS
LIN {X -0.096,Y -208.249,Z 772.159,A 0.000,B 0.000,C 90.000,E1 28.565} C_DIS
LIN {X 0.094,Y -203.275,Z 772.141,A 0.000,B 0.000,C 90.000,E1 25.335} C_DIS
LIN {X -0.038,Y -198.004,Z 772.119,A 0.000,B 0.000,C 90.000,E1 21.354} C_DIS
LIN {X 0.017,Y -193.887,Z 772.096,A 0.000,B 0.000,C 90.000,E1 17.275} C_DIS
LIN {X 0.011,Y -190.287,Z 772.069,A 0.000,B 0.000,C 90.000,E1 12.355} C_DIS
LIN {X 0.014,Y -187.864,Z 772.032,A 0.000,B 0.000,C 90.000,E1 5.739} C_DIS
LIN {X 0.033,Y -189.279,Z 771.970,A 0.000,B 0.000,C 90.000,E1 354.546} C_DIS
LIN {X 0.071,Y -192.764,Z 771.938,A 0.000,B 0.000,C 90.000,E1 348.757} C_DIS
LIN {X -0.009,Y -196.432,Z 771.915,A 0.000,B 0.000,C 90.000,E1 344.685} C_DIS
LIN {X 0.056,Y -201.130,Z 771.892,A 0.000,B 0.000,C 90.000,E1 340.604} C_DIS
LIN {X -0.039,Y -206.819,Z 771.870,A 0.000,B 0.000,C 90.000,E1 336.613} C_DIS
LIN {X 0.078,Y -213.392,Z 771.848,A 0.000,B 0.000,C 90.000,E1 332.615} C_DIS
LIN {X -0.059,Y -220.807,Z 771.826,A 0.000,B 0.000,C 90.000,E1 328.742} C_DIS
LIN {X -0.067,Y -228.811,Z 771.805,A 0.000,B 0.000,C 90.000,E1 324.895} C_DIS
LIN {X 0.023,Y -237.537,Z 771.784,A 0.000,B 0.000,C 90.000,E1 321.090} C_DIS
LIN {X -0.048,Y -247.026,Z 771.763,A 0.000,B 0.000,C 90.000,E1 317.391} C_DIS
LIN {X -0.004,Y -257.420,Z 771.743,A 0.000,B 0.000,C 90.000,E1 313.743} C_DIS
LIN {X -0.024,Y -267.556,Z 771.725,A 0.000,B 0.000,C 90.000,E1 310.539} C_DIS
LIN {X 0.065,Y -279.897,Z 771.706,A 0.000,B 0.000,C 90.000,E1 307.030} C_DIS
LIN {X 0.048,Y -293.479,Z 771.687,A 0.000,B 0.000,C 90.000,E1 303.627} C_DIS
LIN {X 0.036,Y -300.945,Z 771.678,A 0.000,B 0.000,C 90.000,E1 301.957} C_DIS
LIN {X -0.017,Y -317.763,Z 771.659,A 0.000,B 0.000,C 90.000,E1 298.693} C_DIS
LIN {X -0.084,Y -332.317,Z 771.645,A 0.000,B 0.000,C 90.000,E1 296.155} C_DIS
LIN {X -0.062,Y -341.901,Z 771.637,A 0.000,B 0.000,C 90.000,E1 294.591} C_DIS
LIN {X -0.101,Y -358.346,Z 771.623,A 0.000,B 0.000,C 90.000,E1 292.153} C_DIS
LIN {X -0.096,Y -373.851,Z 771.611,A 0.000,B 0.000,C 90.000,E1 290.066} C_DIS
LIN {X -0.217,Y -397.808,Z 771.596,A 0.000,B 0.000,C 90.000,E1 287.221} C_DIS
LIN {X -0.086,Y -412.580,Z 771.586,A 0.000,B 0.000,C 90.000,E1 285.536} C_DIS
LIN {X -0.161,Y -424.676,Z 771.579,A 0.000,B 0.000,C 90.000,E1 284.175} C_DIS
LIN {X -0.162,Y -436.387,Z 771.571,A 0.000,B 0.000,C 90.000,E1 282.827} C_DIS
LIN {X 0.019,Y -447.727,Z 771.564,A 0.000,B 0.000,C 90.000,E1 281.478} C_DIS
LIN {X 0.024,Y -456.196,Z 771.558,A 0.000,B 0.000,C 90.000,E1 280.433} C_DIS
LIN {X -0.036,Y -466.085,Z 771.551,A 0.000,B 0.000,C 90.000,E1 279.151} C_DIS
LIN {X 0.189,Y -473.523,Z 771.545,A 0.000,B 0.000,C 90.000,E1 278.106} C_DIS
LIN {X 0.166,Y -478.580,Z 771.541,A 0.000,B 0.000,C 90.000,E1 277.352} C_DIS
LIN {X 0.122,Y -482.991,Z 771.537,A 0.000,B 0.000,C 90.000,E1 276.606} C_DIS
LIN {X 0.176,Y -486.593,Z 771.533,A 0.000,B 0.000,C 90.000,E1 275.853} C_DIS
LIN {X 0.207,Y -489.419,Z 771.529,A 0.000,B 0.000,C 90.000,E1 275.106} C_DIS
LIN {X -0.072,Y -490.845,Z 771.526,A 0.000,B 0.000,C 90.000,E1 274.645} C_DIS
LIN {X 0.108,Y -491.899,Z 771.523,A 0.000,B 0.000,C 90.000,E1 274.131} C_DIS
LIN {X -0.158,Y -492.575,Z 771.520,A 0.000,B 0.000,C 90.000,E1 273.669} C_DIS
LIN {X 0.044,Y -492.852,Z 771.518,A 0.000,B 0.000,C 90.000,E1 273.154} C_DIS
LIN {X -0.217,Y -492.664,Z 771.515,A 0.000,B 0.000,C 90.000,E1 272.694} C_DIS
LIN {X -0.007,Y -492.081,Z 771.512,A 0.000,B 0.000,C 90.000,E1 272.178} C_DIS
LIN {X 0.218,Y -491.070,Z 771.509,A 0.000,B 0.000,C 90.000,E1 271.661} C_DIS
LIN {X -0.067,Y -489.584,Z 771.507,A 0.000,B 0.000,C 90.000,E1 271.203} C_DIS
LIN {X 0.133,Y -487.546,Z 771.504,A 0.000,B 0.000,C 90.000,E1 270.688} C_DIS
LIN {X -0.161,Y -484.996,Z 771.501,A 0.000,B 0.000,C 90.000,E1 270.229} C_DIS
LIN {X 0.012,Y -481.839,Z 771.498,A 0.000,B 0.000,C 90.000,E1 269.714} C_DIS
LIN {X 0.167,Y -477.885,Z 771.496,A 0.000,B 0.000,C 90.000,E1 269.198} C_DIS
LIN {X -0.175,Y -473.109,Z 771.493,A 0.000,B 0.000,C 90.000,E1 268.740} C_DIS
LIN {X 0.018,Y -467.372,Z 771.490,A 0.000,B 0.000,C 90.000,E1 268.224} C_DIS
LIN {X 0.121,Y -464.420,Z 771.489,A 0.000,B 0.000,C 90.000,E1 267.993} C_DIS
LIN {X 0.127,Y -457.805,Z 771.487,A 0.000,B 0.000,C 90.000,E1 267.593} C_DIS
LIN {X 0.049,Y -454.195,Z 771.486,A 0.000,B 0.000,C 90.000,E1 267.421} C_DIS
LIN {X -0.052,Y -446.743,Z 771.484,A 0.000,B 0.000,C 90.000,E1 267.135} C_DIS
LIN {X -0.083,Y -438.678,Z 771.483,A 0.000,B 0.000,C 90.000,E1 266.906} C_DIS
LIN {X -0.009,Y -429.335,Z 771.482,A 0.000,B 0.000,C 90.000,E1 266.731} C_DIS
LIN {X -0.133,Y -420.638,Z 771.481,A 0.000,B 0.000,C 90.000,E1 266.674} C_DIS
LIN {X -0.186,Y -418.464,Z 771.481,A 0.000,B 0.000,C 90.000,E1 266.674} C_DIS
LIN {X 0.077,Y -180.959,Z 771.481,A 0.000,B 0.000,C 90.000,E1 266.617} C_DIS
LIN {X -0.045,Y -180.883,Z 771.473,A 0.000,B 0.000,C 90.000,E1 265.122} C_DIS
LIN {X 0.076,Y -178.813,Z 771.442,A 0.000,B 0.000,C 90.000,E1 259.511} C_DIS
LIN {X -0.018,Y -175.858,Z 771.414,A 0.000,B 0.000,C 90.000,E1 254.448} C_DIS
LIN {X -0.035,Y -173.187,Z 771.395,A 0.000,B 0.000,C 90.000,E1 251.040} C_DIS
LIN {X -0.034,Y -171.490,Z 771.380,A 0.000,B 0.000,C 90.000,E1 248.465} C_DIS
LIN {X -0.046,Y -167.718,Z 771.356,A 0.000,B 0.000,C 90.000,E1 244.152} C_DIS
LIN {X -0.030,Y -166.411,Z 771.347,A 0.000,B 0.000,C 90.000,E1 242.410} C_DIS
LIN {X -0.031,Y -163.134,Z 771.327,A 0.000,B 0.000,C 90.000,E1 238.918} C_DIS
LIN {X -0.065,Y -161.086,Z 771.313,A 0.000,B 0.000,C 90.000,E1 236.294} C_DIS
LIN {X 0.044,Y -157.816,Z 771.293,A 0.000,B 0.000,C 90.000,E1 232.718} C_DIS
LIN {X -0.018,Y -155.851,Z 771.278,A 0.000,B 0.000,C 90.000,E1 230.070} C_DIS
LIN {X 0.038,Y -152.101,Z 771.253,A 0.000,B 0.000,C 90.000,E1 225.567} C_DIS
LIN {X 0.057,Y -150.352,Z 771.238,A 0.000,B 0.000,C 90.000,E1 222.852} C_DIS
LIN {X -0.014,Y -147.089,Z 771.213,A 0.000,B 0.000,C 90.000,E1 218.338} C_DIS
LIN {X -0.020,Y -145.660,Z 771.198,A 0.000,B 0.000,C 90.000,E1 215.598} C_DIS
LIN {X -0.016,Y -143.042,Z 771.172,A 0.000,B 0.000,C 90.000,E1 211.003} C_DIS
LIN {X -0.015,Y -141.666,Z 771.152,A 0.000,B 0.000,C 90.000,E1 207.308} C_DIS
LIN {X 0.029,Y -139.450,Z 771.116,A 0.000,B 0.000,C 90.000,E1 200.791} C_DIS
LIN {X -0.050,Y -139.184,Z 771.105,A 0.000,B 0.000,C 90.000,E1 198.960} C_DIS
LIN {X -0.027,Y -138.322,Z 771.053,A 0.000,B 0.000,C 90.000,E1 189.613} C_DIS
LIN {X -0.020,Y -139.462,Z 771.007,A 0.000,B 0.000,C 90.000,E1 181.203} C_DIS
LIN {X 0.061,Y -141.021,Z 770.976,A 0.000,B 0.000,C 90.000,E1 175.584} C_DIS
LIN {X 0.015,Y -142.384,Z 770.960,A 0.000,B 0.000,C 90.000,E1 172.818} C_DIS
LIN {X -0.063,Y -144.615,Z 770.934,A 0.000,B 0.000,C 90.000,E1 168.229} C_DIS
LIN {X -0.002,Y -147.809,Z 770.909,A 0.000,B 0.000,C 90.000,E1 163.614} C_DIS
LIN {X 0.085,Y -150.498,Z 770.889,A 0.000,B 0.000,C 90.000,E1 159.934} C_DIS
LIN {X -0.035,Y -153.955,Z 770.869,A 0.000,B 0.000,C 90.000,E1 156.357} C_DIS
LIN {X 0.028,Y -157.366,Z 770.849,A 0.000,B 0.000,C 90.000,E1 152.743} C_DIS
LIN {X -0.030,Y -161.566,Z 770.829,A 0.000,B 0.000,C 90.000,E1 149.203} C_DIS
LIN {X -0.018,Y -165.763,Z 770.809,A 0.000,B 0.000,C 90.000,E1 145.674} C_DIS
LIN {X -0.032,Y -170.720,Z 770.790,A 0.000,B 0.000,C 90.000,E1 142.190} C_DIS
LIN {X 0.012,Y -175.593,Z 770.771,A 0.000,B 0.000,C 90.000,E1 138.728} C_DIS
LIN {X -0.001,Y -181.210,Z 770.752,A 0.000,B 0.000,C 90.000,E1 135.324} C_DIS
LIN {X -0.009,Y -186.675,Z 770.733,A 0.000,B 0.000,C 90.000,E1 131.962} C_DIS
LIN {X -0.005,Y -191.510,Z 770.718,A 0.000,B 0.000,C 90.000,E1 129.322} C_DIS
LIN {X -0.051,Y -192.346,Z 770.716,A 0.000,B 0.000,C 90.000,E1 128.830} C_DIS
LIN {X -0.113,Y -292.019,Z 770.716,A 0.000,B 0.000,C 90.000,E1 128.830} C_DIS
LIN {X 0.010,Y -293.359,Z 770.715,A 0.000,B 0.000,C 90.000,E1 128.785} C_DIS
LIN {X 0.068,Y -297.080,Z 770.715,A 0.000,B 0.000,C 90.000,E1 128.624} C_DIS
LIN {X 0.012,Y -300.328,Z 770.713,A 0.000,B 0.000,C 90.000,E1 128.382} C_DIS
LIN {X -0.060,Y -304.012,Z 770.711,A 0.000,B 0.000,C 90.000,E1 127.935} C_DIS
LIN {X -0.055,Y -305.858,Z 770.709,A 0.000,B 0.000,C 90.000,E1 127.604} C_DIS
LIN {X 0.139,Y -307.299,Z 770.707,A 0.000,B 0.000,C 90.000,E1 127.237} C_DIS
LIN {X 0.132,Y -309.353,Z 770.703,A 0.000,B 0.000,C 90.000,E1 126.583} C_DIS
LIN {X -0.021,Y -319.364,Z 770.685,A 0.000,B 0.000,C 90.000,E1 123.372} C_DIS
LIN {X -0.037,Y -329.688,Z 770.669,A 0.000,B 0.000,C 90.000,E1 120.512} C_DIS
LIN {X -0.146,Y -341.362,Z 770.654,A 0.000,B 0.000,C 90.000,E1 117.719} C_DIS
LIN {X -0.070,Y -354.483,Z 770.639,A 0.000,B 0.000,C 90.000,E1 114.951} C_DIS
LIN {X 0.182,Y -367.459,Z 770.625,A 0.000,B 0.000,C 90.000,E1 112.514} C_DIS
LIN {X 0.147,Y -381.768,Z 770.612,A 0.000,B 0.000,C 90.000,E1 110.174} C_DIS
LIN {X 0.207,Y -397.510,Z 770.599,A 0.000,B 0.000,C 90.000,E1 107.873} C_DIS
LIN {X 0.036,Y -414.799,Z 770.587,A 0.000,B 0.000,C 90.000,E1 105.662} C_DIS
LIN {X 0.079,Y -433.753,Z 770.575,A 0.000,B 0.000,C 90.000,E1 103.480} C_DIS
LIN {X 0.153,Y -453.826,Z 770.564,A 0.000,B 0.000,C 90.000,E1 101.422} C_DIS
LIN {X -0.054,Y -466.668,Z 770.557,A 0.000,B 0.000,C 90.000,E1 100.254} C_DIS
LIN {X -0.007,Y -469.014,Z 770.556,A 0.000,B 0.000,C 90.000,E1 100.018} C_DIS
LIN {X -0.041,Y -470.789,Z 770.554,A 0.000,B 0.000,C 90.000,E1 99.792} C_DIS
LIN {X -0.188,Y -472.278,Z 770.553,A 0.000,B 0.000,C 90.000,E1 99.557} C_DIS
LIN {X 0.129,Y -473.390,Z 770.552,A 0.000,B 0.000,C 90.000,E1 99.265} C_DIS
LIN {X -0.228,Y -474.711,Z 770.549,A 0.000,B 0.000,C 90.000,E1 98.803} C_DIS
LIN {X -0.037,Y -475.016,Z 770.546,A 0.000,B 0.000,C 90.000,E1 98.276} C_DIS
LIN {X 0.090,Y -474.357,Z 770.543,A 0.000,B 0.000,C 90.000,E1 97.757} C_DIS
LIN {X 0.220,Y -472.632,Z 770.540,A 0.000,B 0.000,C 90.000,E1 97.239} C_DIS
LIN {X 0.078,Y -471.271,Z 770.539,A 0.000,B 0.000,C 90.000,E1 97.004} C_DIS
LIN {X -0.017,Y -451.905,Z 770.522,A 0.000,B 0.000,C 90.000,E1 93.955} C_DIS
LIN {X -0.193,Y -439.941,Z 770.510,A 0.000,B 0.000,C 90.000,E1 91.892} C_DIS
LIN {X -0.061,Y -430.724,Z 770.502,A 0.000,B 0.000,C 90.000,E1 90.286} C_DIS
LIN {X -0.102,Y -421.195,Z 770.493,A 0.000,B 0.000,C 90.000,E1 88.682} C_DIS
LIN {X -0.191,Y -410.009,Z 770.482,A 0.000,B 0.000,C 90.000,E1 86.788} C_DIS
LIN {X -0.104,Y -398.621,Z 770.471,A 0.000,B 0.000,C 90.000,E1 84.837} C_DIS
LIN {X -0.177,Y -387.353,Z 770.460,A 0.000,B 0.000,C 90.000,E1 82.875} C_DIS
LIN {X -0.090,Y -373.243,Z 770.446,A 0.000,B 0.000,C 90.000,E1 80.274} C_DIS
LIN {X 0.161,Y -356.816,Z 770.428,A 0.000,B 0.000,C 90.000,E1 76.992} C_DIS
LIN {X -0.156,Y -346.792,Z 770.416,A 0.000,B 0.000,C 90.000,E1 74.936} C_DIS
LIN {X -0.082,Y -335.469,Z 770.403,A 0.000,B 0.000,C 90.000,E1 72.472} C_DIS
LIN {X -0.014,Y -323.073,Z 770.387,A 0.000,B 0.000,C 90.000,E1 69.645} C_DIS
LIN {X 0.098,Y -308.723,Z 770.367,A 0.000,B 0.000,C 90.000,E1 66.102} C_DIS
LIN {X 0.117,Y -295.661,Z 770.347,A 0.000,B 0.000,C 90.000,E1 62.487} C_DIS
LIN {X 0.059,Y -287.011,Z 770.332,A 0.000,B 0.000,C 90.000,E1 59.822} C_DIS
LIN {X 0.054,Y -276.850,Z 770.314,A 0.000,B 0.000,C 90.000,E1 56.421} C_DIS
LIN {X 0.037,Y -268.955,Z 770.298,A 0.000,B 0.000,C 90.000,E1 53.657} C_DIS
LIN {X -0.129,Y -261.097,Z 770.283,A 0.000,B 0.000,C 90.000,E1 50.884} C_DIS
LIN {X 0.014,Y -253.317,Z 770.267,A 0.000,B 0.000,C 90.000,E1 48.000} C_DIS
LIN {X 0.112,Y -245.658,Z 770.251,A 0.000,B 0.000,C 90.000,E1 45.081} C_DIS
LIN {X -0.112,Y -240.036,Z 770.238,A 0.000,B 0.000,C 90.000,E1 42.933} C_DIS
LIN {X 0.007,Y -232.585,Z 770.222,A 0.000,B 0.000,C 90.000,E1 39.930} C_DIS
LIN {X -0.077,Y -223.741,Z 770.201,A 0.000,B 0.000,C 90.000,E1 36.171} C_DIS
LIN {X 0.036,Y -215.518,Z 770.179,A 0.000,B 0.000,C 90.000,E1 32.291} C_DIS
LIN {X 0.064,Y -209.635,Z 770.162,A 0.000,B 0.000,C 90.000,E1 29.155} C_DIS
LIN {X 0.104,Y -204.489,Z 770.144,A 0.000,B 0.000,C 90.000,E1 25.976} C_DIS
LIN {X -0.097,Y -199.009,Z 770.122,A 0.000,B 0.000,C 90.000,E1 22.025} C_DIS
LIN {X -0.010,Y -194.702,Z 770.100,A 0.000,B 0.000,C 90.000,E1 17.946} C_DIS
LIN {X 0.077,Y -191.411,Z 770.077,A 0.000,B 0.000,C 90.000,E1 13.828} C_DIS
LIN {X -0.094,Y -188.609,Z 770.045,A 0.000,B 0.000,C 90.000,E1 8.106} C_DIS
LIN {X -0.039,Y -189.797,Z 769.965,A 0.000,B 0.000,C 90.000,E1 353.742} C_DIS
LIN {X 0.081,Y -192.885,Z 769.938,A 0.000,B 0.000,C 90.000,E1 348.757} C_DIS
LIN {X 0.005,Y -196.557,Z 769.915,A 0.000,B 0.000,C 90.000,E1 344.685} C_DIS
LIN {X 0.075,Y -201.274,Z 769.892,A 0.000,B 0.000,C 90.000,E1 340.604} C_DIS
LIN {X -0.015,Y -206.955,Z 769.870,A 0.000,B 0.000,C 90.000,E1 336.613} C_DIS
LIN {X 0.107,Y -213.517,Z 769.848,A 0.000,B 0.000,C 90.000,E1 332.615} C_DIS
LIN {X -0.026,Y -220.918,Z 769.826,A 0.000,B 0.000,C 90.000,E1 328.742} C_DIS
LIN {X -0.030,Y -228.908,Z 769.805,A 0.000,B 0.000,C 90.000,E1 324.895} C_DIS
LIN {X 0.066,Y -237.616,Z 769.784,A 0.000,B 0.000,C 90.000,E1 321.090} C_DIS
LIN {X -0.001,Y -247.072,Z 769.763,A 0.000,B 0.000,C 90.000,E1 317.391} C_DIS
LIN {X -0.140,Y -257.450,Z 769.743,A 0.000,B 0.000,C 90.000,E1 313.785} C_DIS
LIN {X 0.029,Y -267.571,Z 769.725,A 0.000,B 0.000,C 90.000,E1 310.539} C_DIS
LIN {X -0.102,Y -279.908,Z 769.706,A 0.000,B 0.000,C 90.000,E1 307.076} C_DIS
LIN {X -0.056,Y -293.454,Z 769.687,A 0.000,B 0.000,C 90.000,E1 303.658} C_DIS
LIN {X -0.159,Y -300.915,Z 769.678,A 0.000,B 0.000,C 90.000,E1 302.005} C_DIS
LIN {X 0.045,Y -317.723,Z 769.659,A 0.000,B 0.000,C 90.000,E1 298.693} C_DIS
LIN {X -0.054,Y -334.096,Z 769.644,A 0.000,B 0.000,C 90.000,E1 295.848} C_DIS
LIN {X 0.137,Y -343.822,Z 769.635,A 0.000,B 0.000,C 90.000,E1 294.259} C_DIS
LIN {X 0.128,Y -364.710,Z 769.618,A 0.000,B 0.000,C 90.000,E1 291.227} C_DIS
LIN {X 0.055,Y -387.885,Z 769.602,A 0.000,B 0.000,C 90.000,E1 288.308} C_DIS
LIN {X -0.091,Y -402.781,Z 769.592,A 0.000,B 0.000,C 90.000,E1 286.622} C_DIS
LIN {X -0.090,Y -414.989,Z 769.585,A 0.000,B 0.000,C 90.000,E1 285.245} C_DIS
LIN {X -0.140,Y -427.011,Z 769.577,A 0.000,B 0.000,C 90.000,E1 283.883} C_DIS
LIN {X -0.103,Y -438.608,Z 769.570,A 0.000,B 0.000,C 90.000,E1 282.535} C_DIS
LIN {X -0.121,Y -447.648,Z 769.564,A 0.000,B 0.000,C 90.000,E1 281.478} C_DIS
LIN {X -0.038,Y -456.074,Z 769.558,A 0.000,B 0.000,C 90.000,E1 280.423} C_DIS
LIN {X -0.186,Y -465.994,Z 769.551,A 0.000,B 0.000,C 90.000,E1 279.151} C_DIS
LIN {X 0.036,Y -473.436,Z 769.545,A 0.000,B 0.000,C 90.000,E1 278.106} C_DIS
LIN {X 0.011,Y -478.548,Z 769.541,A 0.000,B 0.000,C 90.000,E1 277.352} C_DIS
LIN {X -0.036,Y -482.984,Z 769.537,A 0.000,B 0.000,C 90.000,E1 276.606} C_DIS
LIN {X 0.018,Y -486.620,Z 769.533,A 0.000,B 0.000,C 90.000,E1 275.853} C_DIS
LIN {X 0.049,Y -489.460,Z 769.528,A 0.000,B 0.000,C 90.000,E1 275.106} C_DIS
LIN {X -0.232,Y -490.874,Z 769.526,A 0.000,B 0.000,C 90.000,E1 274.645} C_DIS
LIN {X -0.051,Y -491.984,Z 769.523,A 0.000,B 0.000,C 90.000,E1 274.131} C_DIS
LIN {X 0.174,Y -492.645,Z 769.520,A 0.000,B 0.000,C 90.000,E1 273.612} C_DIS
LIN {X -0.116,Y -492.938,Z 769.517,A 0.000,B 0.000,C 90.000,E1 273.154} C_DIS
LIN {X 0.116,Y -492.785,Z 769.515,A 0.000,B 0.000,C 90.000,E1 272.636} C_DIS
LIN {X -0.165,Y -492.209,Z 769.512,A 0.000,B 0.000,C 90.000,E1 272.178} C_DIS
LIN {X 0.061,Y -491.193,Z 769.509,A 0.000,B 0.000,C 90.000,E1 271.661} C_DIS
LIN {X -0.223,Y -489.705,Z 769.507,A 0.000,B 0.000,C 90.000,E1 271.203} C_DIS
LIN {X -0.022,Y -487.663,Z 769.504,A 0.000,B 0.000,C 90.000,E1 270.688} C_DIS
LIN {X 0.171,Y -485.094,Z 769.501,A 0.000,B 0.000,C 90.000,E1 270.172} C_DIS
LIN {X -0.138,Y -481.909,Z 769.498,A 0.000,B 0.000,C 90.000,E1 269.714} C_DIS
LIN {X 0.017,Y -477.983,Z 769.496,A 0.000,B 0.000,C 90.000,E1 269.198} C_DIS
LIN {X 0.150,Y -473.143,Z 769.493,A 0.000,B 0.000,C 90.000,E1 268.682} C_DIS
LIN {X -0.117,Y -467.397,Z 769.490,A 0.000,B 0.000,C 90.000,E1 268.224} C_DIS
LIN {X -0.006,Y -464.420,Z 769.489,A 0.000,B 0.000,C 90.000,E1 267.993} C_DIS
LIN {X 0.013,Y -457.847,Z 769.487,A 0.000,B 0.000,C 90.000,E1 267.593} C_DIS
LIN {X 0.125,Y -450.761,Z 769.485,A 0.000,B 0.000,C 90.000,E1 267.249} C_DIS
LIN {X -0.152,Y -443.222,Z 769.483,A 0.000,B 0.000,C 90.000,E1 267.020} C_DIS
LIN {X 0.112,Y -434.796,Z 769.482,A 0.000,B 0.000,C 90.000,E1 266.788} C_DIS
LIN {X 0.022,Y -425.807,Z 769.482,A 0.000,B 0.000,C 90.000,E1 266.674} C_DIS
LIN {X 0.110,Y -415.879,Z 769.481,A 0.000,B 0.000,C 90.000,E1 266.617} C_DIS
LIN {X 0.024,Y -180.958,Z 769.481,A 0.000,B 0.000,C 90.000,E1 266.617} C_DIS
LIN {X -0.076,Y -180.882,Z 769.473,A 0.000,B 0.000,C 90.000,E1 265.122} C_DIS
LIN {X 0.046,Y -178.809,Z 769.442,A 0.000,B 0.000,C 90.000,E1 259.511} C_DIS
LIN {X -0.048,Y -175.853,Z 769.414,A 0.000,B 0.000,C 90.000,E1 254.448} C_DIS
LIN {X -0.066,Y -173.181,Z 769.395,A 0.000,B 0.000,C 90.000,E1 251.040} C_DIS
LIN {X -0.064,Y -171.481,Z 769.380,A 0.000,B 0.000,C 90.000,E1 248.465} C_DIS
LIN {X -0.076,Y -167.711,Z 769.356,A 0.000,B 0.000,C 90.000,E1 244.152} C_DIS
LIN {X -0.059,Y -166.400,Z 769.347,A 0.000,B 0.000,C 90.000,E1 242.410} C_DIS
LIN {X 0.079,Y -163.126,Z 769.327,A 0.000,B 0.000,C 90.000,E1 238.869} C_DIS
LIN {X -0.094,Y -161.077,Z 769.313,A 0.000,B 0.000,C 90.000,E1 236.294} C_DIS
LIN {X 0.016,Y -157.808,Z 769.293,A 0.000,B 0.000,C 90.000,E1 232.718} C_DIS
LIN {X -0.046,Y -155.843,Z 769.278,A 0.000,B 0.000,C 90.000,E1 230.070} C_DIS
LIN {X 0.010,Y -152.093,Z 769.253,A 0.000,B 0.000,C 90.000,E1 225.567} C_DIS
LIN {X 0.029,Y -150.344,Z 769.238,A 0.000,B 0.000,C 90.000,E1 222.852} C_DIS
LIN {X 0.050,Y -147.081,Z 769.213,A 0.000,B 0.000,C 90.000,E1 218.302} C_DIS
LIN {X -0.047,Y -145.655,Z 769.198,A 0.000,B 0.000,C 90.000,E1 215.598} C_DIS
LIN {X -0.043,Y -143.037,Z 769.172,A 0.000,B 0.000,C 90.000,E1 211.003} C_DIS
LIN {X -0.042,Y -141.661,Z 769.152,A 0.000,B 0.000,C 90.000,E1 207.308} C_DIS
LIN {X 0.003,Y -139.449,Z 769.116,A 0.000,B 0.000,C 90.000,E1 200.791} C_DIS
LIN {X 0.056,Y -139.182,Z 769.105,A 0.000,B 0.000,C 90.000,E1 198.906} C_DIS
LIN {X -0.053,Y -138.320,Z 769.053,A 0.000,B 0.000,C 90.000,E1 189.613} C_DIS
LIN {X -0.046,Y -139.464,Z 769.007,A 0.000,B 0.000,C 90.000,E1 181.203} C_DIS
LIN {X 0.034,Y -141.025,Z 768.976,A 0.000,B 0.000,C 90.000,E1 175.584} C_DIS
LIN {X -0.011,Y -142.391,Z 768.960,A 0.000,B 0.000,C 90.000,E1 172.818} C_DIS
LIN {X 0.052,Y -144.621,Z 768.934,A 0.000,B 0.000,C 90.000,E1 168.173} C_DIS
LIN {X -0.029,Y -147.816,Z 768.909,A 0.000,B 0.000,C 90.000,E1 163.614} C_DIS
LIN {X 0.057,Y -150.506,Z 768.889,A 0.000,B 0.000,C 90.000,E1 159.934} C_DIS
LIN {X -0.063,Y -153.965,Z 768.869,A 0.000,B 0.000,C 90.000,E1 156.357} C_DIS
LIN {X 0.000,Y -157.377,Z 768.849,A 0.000,B 0.000,C 90.000,E1 152.743} C_DIS
LIN {X -0.059,Y -161.579,Z 768.829,A 0.000,B 0.000,C 90.000,E1 149.203} C_DIS
LIN {X -0.047,Y -165.776,Z 768.809,A 0.000,B 0.000,C 90.000,E1 145.674} C_DIS
LIN {X -0.061,Y -170.735,Z 768.790,A 0.000,B 0.000,C 90.000,E1 142.190} C_DIS
LIN {X -0.019,Y -175.608,Z 768.771,A 0.000,B 0.000,C 90.000,E1 138.728} C_DIS
LIN {X -0.033,Y -181.224,Z 768.752,A 0.000,B 0.000,C 90.000,E1 135.324} C_DIS
LIN {X 0.099,Y -186.691,Z 768.733,A 0.000,B 0.000,C 90.000,E1 131.919} C_DIS
LIN {X -0.036,Y -191.525,Z 768.718,A 0.000,B 0.000,C 90.000,E1 129.322} C_DIS
LIN {X 0.013,Y -192.314,Z 768.716,A 0.000,B 0.000,C 90.000,E1 128.830} C_DIS
LIN {X -0.015,Y -292.027,Z 768.716,A 0.000,B 0.000,C 90.000,E1 128.830} C_DIS
LIN {X -0.121,Y -293.312,Z 768.716,A 0.000,B 0.000,C 90.000,E1 128.830} C_DIS
LIN {X 0.018,Y -297.473,Z 768.715,A 0.000,B 0.000,C 90.000,E1 128.624} C_DIS
LIN {X -0.121,Y -300.695,Z 768.713,A 0.000,B 0.000,C 90.000,E1 128.382} C_DIS
LIN {X -0.102,Y -304.380,Z 768.710,A 0.000,B 0.000,C 90.000,E1 127.890} C_DIS
LIN {X 0.092,Y -306.125,Z 768.709,A 0.000,B 0.000,C 90.000,E1 127.523} C_DIS
LIN {X -0.144,Y -307.493,Z 768.707,A 0.000,B 0.000,C 90.000,E1 127.237} C_DIS
LIN {X -0.045,Y -315.329,Z 768.692,A 0.000,B 0.000,C 90.000,E1 124.612} C_DIS
LIN {X 0.090,Y -326.274,Z 768.674,A 0.000,B 0.000,C 90.000,E1 121.386} C_DIS
LIN {X 0.055,Y -337.511,Z 768.659,A 0.000,B 0.000,C 90.000,E1 118.565} C_DIS
LIN {X 0.029,Y -350.166,Z 768.643,A 0.000,B 0.000,C 90.000,E1 115.796} C_DIS
LIN {X -0.006,Y -362.693,Z 768.630,A 0.000,B 0.000,C 90.000,E1 113.387} C_DIS
LIN {X -0.164,Y -376.518,Z 768.617,A 0.000,B 0.000,C 90.000,E1 111.046} C_DIS
LIN {X -0.110,Y -391.740,Z 768.604,A 0.000,B 0.000,C 90.000,E1 108.725} C_DIS
LIN {X 0.077,Y -408.468,Z 768.591,A 0.000,B 0.000,C 90.000,E1 106.441} C_DIS
LIN {X 0.064,Y -426.823,Z 768.579,A 0.000,B 0.000,C 90.000,E1 104.245} C_DIS
LIN {X 0.210,Y -446.634,Z 768.568,A 0.000,B 0.000,C 90.000,E1 102.119} C_DIS
LIN {X 0.089,Y -467.071,Z 768.557,A 0.000,B 0.000,C 90.000,E1 100.197} C_DIS
LIN {X 0.140,Y -469.326,Z 768.555,A 0.000,B 0.000,C 90.000,E1 99.962} C_DIS
LIN {X 0.191,Y -471.029,Z 768.554,A 0.000,B 0.000,C 90.000,E1 99.726} C_DIS
LIN {X -0.035,Y -472.462,Z 768.553,A 0.000,B 0.000,C 90.000,E1 99.500} C_DIS
LIN {X -0.183,Y -473.528,Z 768.551,A 0.000,B 0.000,C 90.000,E1 99.265} C_DIS
LIN {X -0.070,Y -474.777,Z 768.549,A 0.000,B 0.000,C 90.000,E1 98.746} C_DIS
LIN {X 0.121,Y -475.019,Z 768.546,A 0.000,B 0.000,C 90.000,E1 98.219} C_DIS
LIN {X -0.221,Y -474.294,Z 768.543,A 0.000,B 0.000,C 90.000,E1 97.757} C_DIS
LIN {X -0.089,Y -472.488,Z 768.540,A 0.000,B 0.000,C 90.000,E1 97.239} C_DIS
LIN {X 0.237,Y -471.075,Z 768.539,A 0.000,B 0.000,C 90.000,E1 96.947} C_DIS
